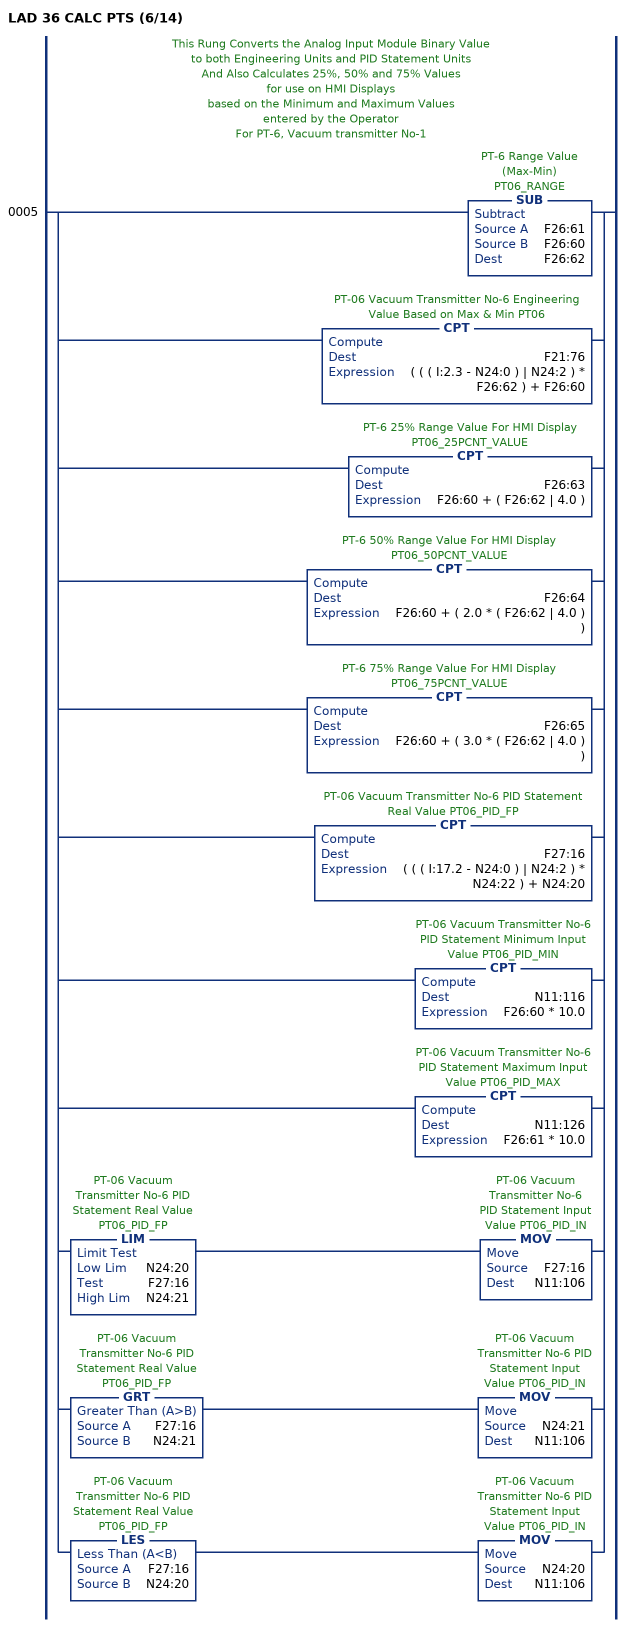
% Rung: 5 %
% This Rung Converts the Analog Input Module Binary Value
% to both Engineering Units and PID Statement Units
% And Also Calculates 25%, 50% and 75% Values
% for use on HMI Displays
% based on the Minimum and Maximum Values
% entered by the Operator
%    For PT-6, Vacuum transmitter No-1 %
SOR BST SUB F26:61 F26:60 F26:62 NXB CPT F21:76 " ( ( ( I:2.3 - N24:0 ) | N24:2 ) * F26:62 ) + F26:60 " NXB CPT F26:63 " F26:60 + ( F26:62 | 4.0 ) " NXB CPT F26:64 " F26:60 + ( 2.0 * ( F26:62 | 4.0 ) ) " NXB CPT F26:65 " F26:60 + ( 3.0 * ( F26:62 | 4.0 ) ) " NXB CPT F27:16 " ( ( ( I:17.2 - N24:0 ) | N24:2 ) * N24:22 ) + N24:20 " NXB CPT N11:116 " F26:60 * 10.0 " NXB CPT N11:126 " F26:61 * 10.0 " NXB LIM N24:20 F27:16 N24:21 MOV F27:16 N11:106 NXB GRT F27:16 N24:21 MOV N24:21 N11:106 NXB LES F27:16 N24:20 MOV N24:20 N11:106 BND EOR
%   F26:61  PT06_MAX  "PT-6 Maximum Value" %
%   F26:60  PT06_MIN  "PT-6 Minimum Value" %
%   F26:62  PT06_RANGE  "PT-6 Range Value (Max-Min)" %
%   F21:76  PT06  "PT-06 Vacuum Transmitter No-6 Engineering Value Based on Max & Min" %
%   I:2.3  PT61_BIN  "PT-6 Binary Input From Transmitter Analog Input Module" %
%   N24:0  AI_CURRENT_MIN  "Analog Input Minimum Value = 4 mA DC (From AI Module)" %
%   N24:2  AI_CURRENT_RANGE  "Analog Input Current Range Value = (AI_MAX - AI_MIN) For Use Elswhere" %
%   F26:63  PT06_25PCNT_VALUE  "PT-6 25% Range Value For HMI Display" %
%   F26:64  PT06_50PCNT_VALUE  "PT-6 50% Range Value For HMI Display" %
%   F26:65  PT06_75PCNT_VALUE  "PT-6 75% Range Value For HMI Display" %
%   F27:16  PT06_PID_FP  "PT-06 Vacuum Transmitter No-6 PID Statement Real Value" %
%   I:17.2  FT06_BIN  "FT-6 Feed Flow Binary Input From Transmitter 1 Analog Input Module" %
%   N24:22  PID_RANGE  "PID Statement Range Value = (PID_MAX - PID_MIN) For Use Elswhere" %
%   N24:20  PID_MIN  "PID Statement Minimum Value" %
%   N11:116  PT06_PID_MIN  "PT-06 Vacuum Transmitter No-6 PID Statement Minimum Input Value" %
%   N11:126  PT06_PID_MAX  "PT-06 Vacuum Transmitter No-6 PID Statement Maximum Input Value" %
%   N24:21  PID_MAX  "PID Statement Maximum Value" %
%   N11:106  PT06_PID_IN  "PT-06 Vacuum Transmitter No-6 PID Statement Input Value" %

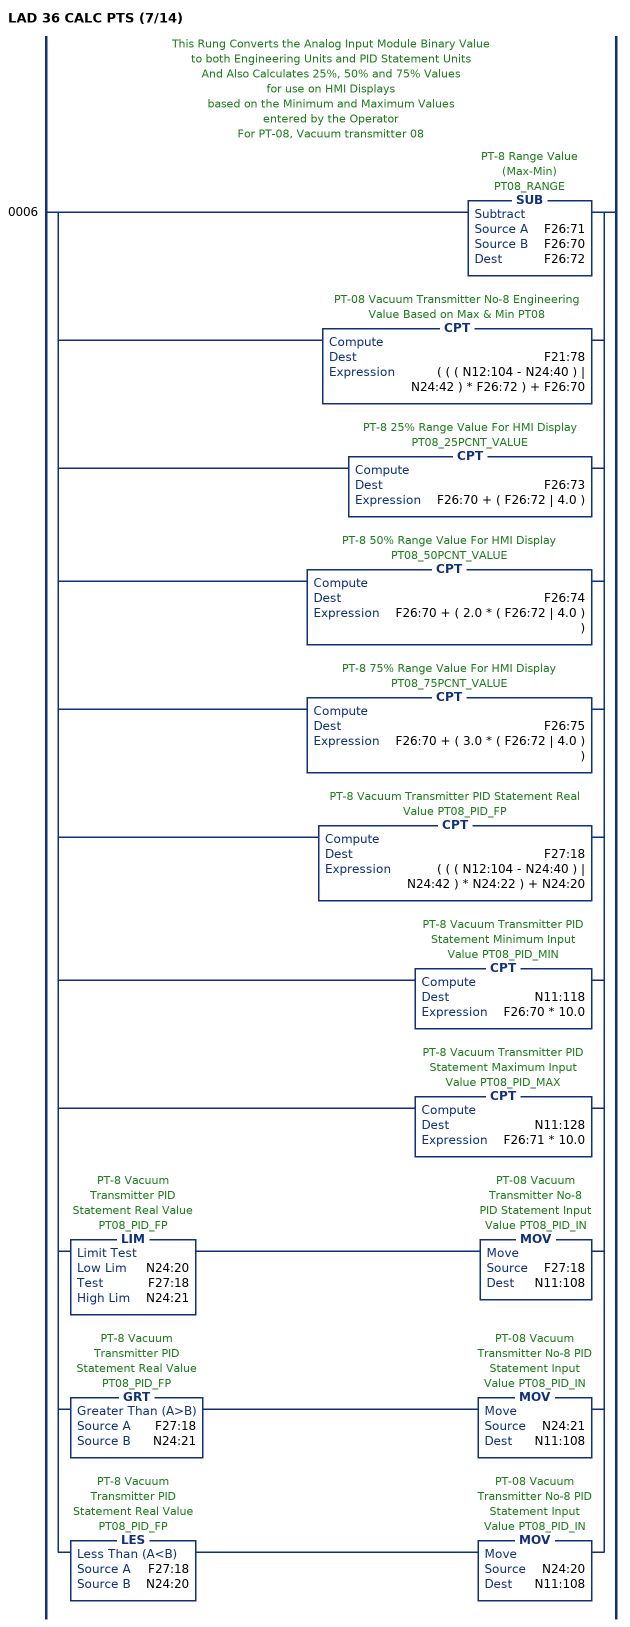
% Rung: 6 %
% This Rung Converts the Analog Input Module Binary Value
% to both Engineering Units and PID Statement Units
% And Also Calculates 25%, 50% and 75% Values
% for use on HMI Displays
% based on the Minimum and Maximum Values
% entered by the Operator
%    For PT-08, Vacuum transmitter 08 %
SOR BST SUB F26:71 F26:70 F26:72 NXB CPT F21:78 " ( ( ( N12:104 - N24:40 ) | N24:42 ) * F26:72 ) + F26:70 " NXB CPT F26:73 " F26:70 + ( F26:72 | 4.0 ) " NXB CPT F26:74 " F26:70 + ( 2.0 * ( F26:72 | 4.0 ) ) " NXB CPT F26:75 " F26:70 + ( 3.0 * ( F26:72 | 4.0 ) ) " NXB CPT F27:18 " ( ( ( N12:104 - N24:40 ) | N24:42 ) * N24:22 ) + N24:20 " NXB CPT N11:118 " F26:70 * 10.0 " NXB CPT N11:128 " F26:71 * 10.0 " NXB LIM N24:20 F27:18 N24:21 MOV F27:18 N11:108 NXB GRT F27:18 N24:21 MOV N24:21 N11:108 NXB LES F27:18 N24:20 MOV N24:20 N11:108 BND EOR
%   F26:71  PT08_MAX  "PT-8 Maximum Value" %
%   F26:70  PT08_MIN  "PT-8 Minimum Value" %
%   F26:72  PT08_RANGE  "PT-8 Range Value (Max-Min)" %
%   F21:78  PT08  "PT-08 Vacuum Transmitter No-8 Engineering Value Based on Max & Min" %
%   N12:104  AI105_BIN_DATA %
%   N24:40  AI_CURRENT_MIN_IE8  "Analog Input Minimum Value = 4 mA DC (From IE8 AI Module)" %
%   N24:42  AI_CURRENT_RANGE_IE8  "IE8 Analog Input Current Range Value = (AI_MAX - AI_MIN) For Use Elswhere" %
%   F26:73  PT08_25PCNT_VALUE  "PT-8 25% Range Value For HMI Display" %
%   F26:74  PT08_50PCNT_VALUE  "PT-8 50% Range Value For HMI Display" %
%   F26:75  PT08_75PCNT_VALUE  "PT-8 75% Range Value For HMI Display" %
%   F27:18  PT08_PID_FP  "PT-8 Vacuum Transmitter PID Statement Real Value" %
%   N24:22  PID_RANGE  "PID Statement Range Value = (PID_MAX - PID_MIN) For Use Elswhere" %
%   N24:20  PID_MIN  "PID Statement Minimum Value" %
%   N11:118  PT08_PID_MIN  "PT-8 Vacuum Transmitter PID Statement Minimum Input Value" %
%   N11:128  PT08_PID_MAX  "PT-8 Vacuum Transmitter PID Statement Maximum Input Value" %
%   N24:21  PID_MAX  "PID Statement Maximum Value" %
%   N11:108  PT08_PID_IN  "PT-08 Vacuum Transmitter No-8 PID Statement Input Value" %

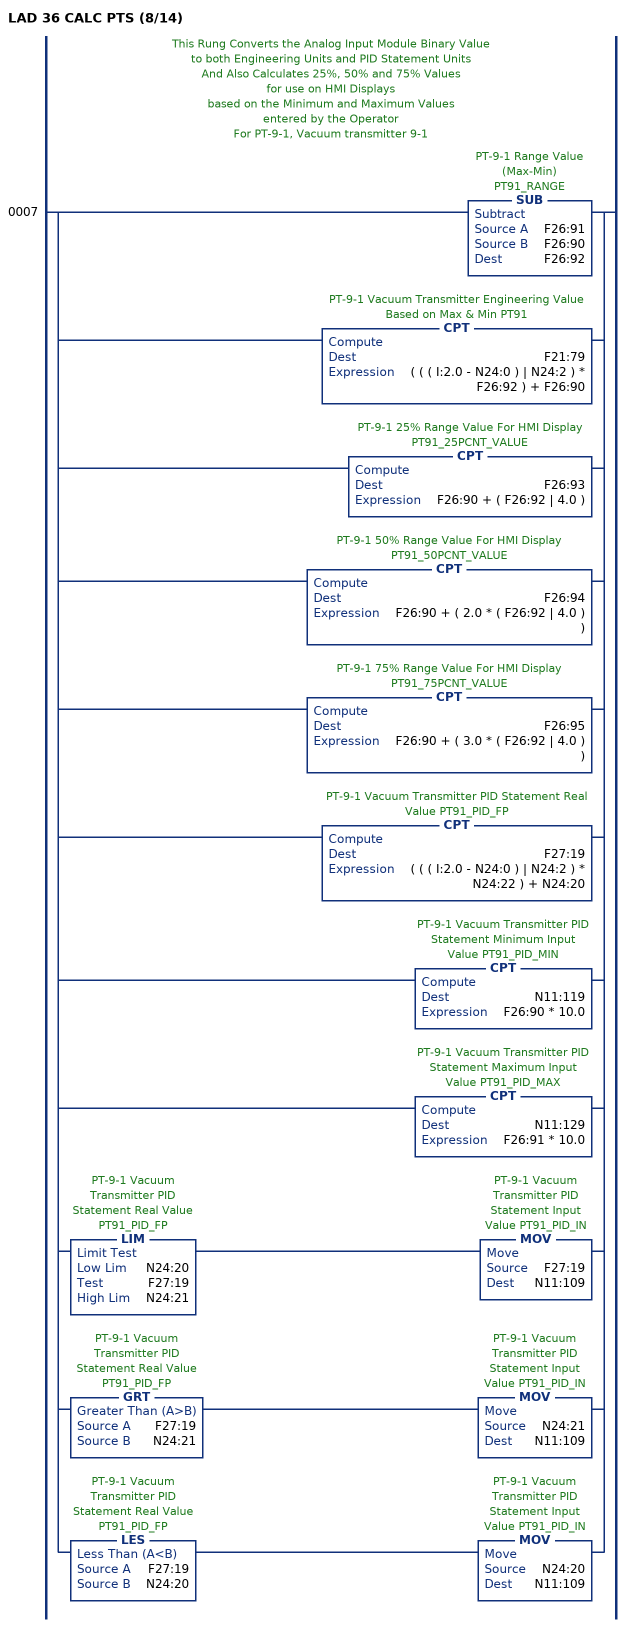
% Rung: 7 %
% This Rung Converts the Analog Input Module Binary Value
% to both Engineering Units and PID Statement Units
% And Also Calculates 25%, 50% and 75% Values
% for use on HMI Displays
% based on the Minimum and Maximum Values
% entered by the Operator
%    For PT-9-1, Vacuum transmitter 9-1 %
SOR BST SUB F26:91 F26:90 F26:92 NXB CPT F21:79 " ( ( ( I:2.0 - N24:0 ) | N24:2 ) * F26:92 ) + F26:90 " NXB CPT F26:93 " F26:90 + ( F26:92 | 4.0 ) " NXB CPT F26:94 " F26:90 + ( 2.0 * ( F26:92 | 4.0 ) ) " NXB CPT F26:95 " F26:90 + ( 3.0 * ( F26:92 | 4.0 ) ) " NXB CPT F27:19 " ( ( ( I:2.0 - N24:0 ) | N24:2 ) * N24:22 ) + N24:20 " NXB CPT N11:119 " F26:90 * 10.0 " NXB CPT N11:129 " F26:91 * 10.0 " NXB LIM N24:20 F27:19 N24:21 MOV F27:19 N11:109 NXB GRT F27:19 N24:21 MOV N24:21 N11:109 NXB LES F27:19 N24:20 MOV N24:20 N11:109 BND EOR
%   F26:91  PT91_MAX  "PT-9-1 Maximum Value" %
%   F26:90  PT91_MIN  "PT-9-1 Minimum Value" %
%   F26:92  PT91_RANGE  "PT-9-1 Range Value (Max-Min)" %
%   F21:79  PT91  "PT-9-1 Vacuum Transmitter Engineering Value Based on Max & Min" %
%   I:2.0  PT91_BIN  "PT-9-1 Binary Input From Transmitter Analog Input Module" %
%   N24:0  AI_CURRENT_MIN  "Analog Input Minimum Value = 4 mA DC (From AI Module)" %
%   N24:2  AI_CURRENT_RANGE  "Analog Input Current Range Value = (AI_MAX - AI_MIN) For Use Elswhere" %
%   F26:93  PT91_25PCNT_VALUE  "PT-9-1 25% Range Value For HMI Display" %
%   F26:94  PT91_50PCNT_VALUE  "PT-9-1 50% Range Value For HMI Display" %
%   F26:95  PT91_75PCNT_VALUE  "PT-9-1 75% Range Value For HMI Display" %
%   F27:19  PT91_PID_FP  "PT-9-1 Vacuum Transmitter PID Statement Real Value" %
%   N24:22  PID_RANGE  "PID Statement Range Value = (PID_MAX - PID_MIN) For Use Elswhere" %
%   N24:20  PID_MIN  "PID Statement Minimum Value" %
%   N11:119  PT91_PID_MIN  "PT-9-1 Vacuum Transmitter PID Statement Minimum Input Value" %
%   N11:129  PT91_PID_MAX  "PT-9-1 Vacuum Transmitter PID Statement Maximum Input Value" %
%   N24:21  PID_MAX  "PID Statement Maximum Value" %
%   N11:109  PT91_PID_IN  "PT-9-1 Vacuum Transmitter PID Statement Input Value" %

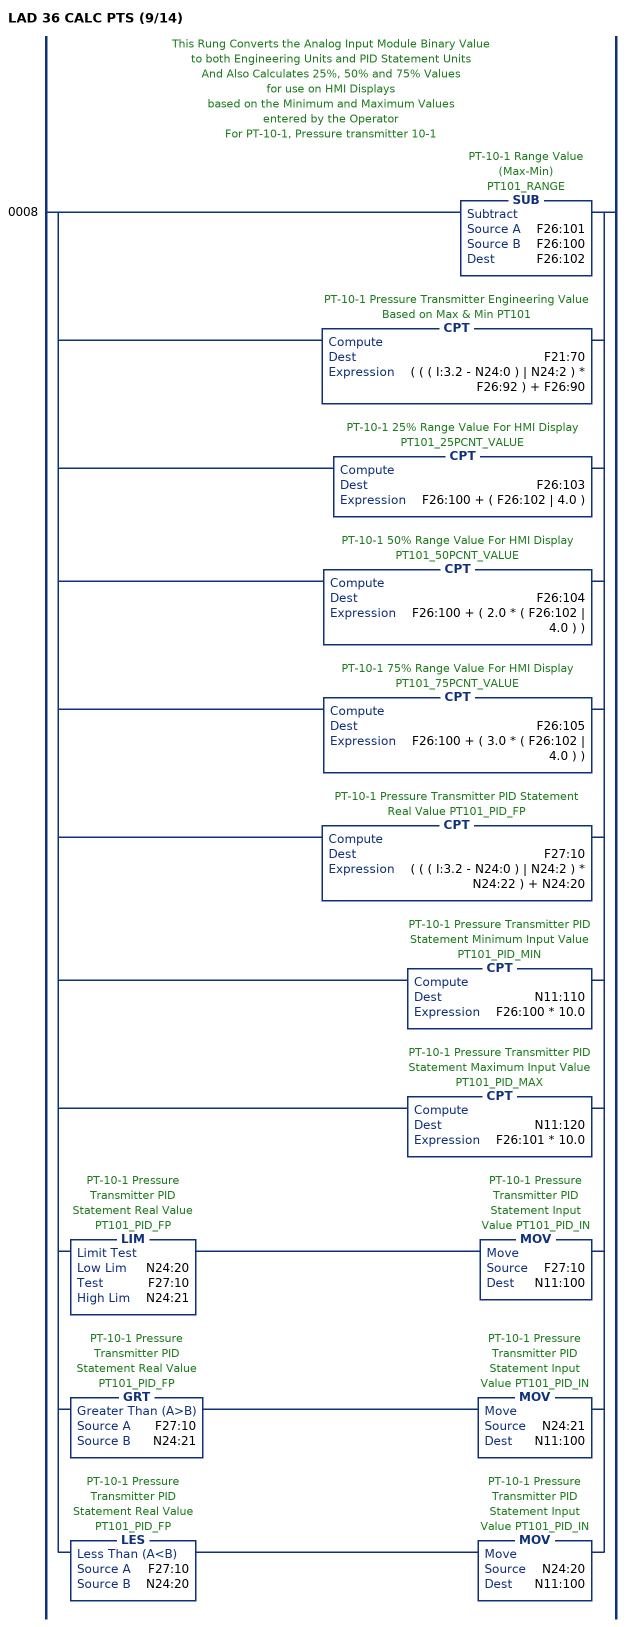
% Rung: 8 %
% This Rung Converts the Analog Input Module Binary Value
% to both Engineering Units and PID Statement Units
% And Also Calculates 25%, 50% and 75% Values
% for use on HMI Displays
% based on the Minimum and Maximum Values
% entered by the Operator
%    For PT-10-1, Pressure transmitter 10-1 %
SOR BST SUB F26:101 F26:100 F26:102 NXB CPT F21:70 " ( ( ( I:3.2 - N24:0 ) | N24:2 ) * F26:92 ) + F26:90 " NXB CPT F26:103 " F26:100 + ( F26:102 | 4.0 ) " NXB CPT F26:104 " F26:100 + ( 2.0 * ( F26:102 | 4.0 ) ) " NXB CPT F26:105 " F26:100 + ( 3.0 * ( F26:102 | 4.0 ) ) " NXB CPT F27:10 " ( ( ( I:3.2 - N24:0 ) | N24:2 ) * N24:22 ) + N24:20 " NXB CPT N11:110 " F26:100 * 10.0 " NXB CPT N11:120 " F26:101 * 10.0 " NXB LIM N24:20 F27:10 N24:21 MOV F27:10 N11:100 NXB GRT F27:10 N24:21 MOV N24:21 N11:100 NXB LES F27:10 N24:20 MOV N24:20 N11:100 BND EOR
%   F26:101  PT101_MAX  "PT-10-1 Maximum Value" %
%   F26:100  PT101_MIN  "PT-10-1 Minimum Value" %
%   F26:102  PT101_RANGE  "PT-10-1 Range Value (Max-Min)" %
%   F21:70  PT101  "PT-10-1 Pressure Transmitter Engineering Value Based on Max & Min" %
%   I:3.2  PT101_BIN  "PT-10-1 Press Binary Input From Transmitter Analog Input Module" %
%   N24:0  AI_CURRENT_MIN  "Analog Input Minimum Value = 4 mA DC (From AI Module)" %
%   N24:2  AI_CURRENT_RANGE  "Analog Input Current Range Value = (AI_MAX - AI_MIN) For Use Elswhere" %
%   F26:92  PT91_RANGE  "PT-9-1 Range Value (Max-Min)" %
%   F26:90  PT91_MIN  "PT-9-1 Minimum Value" %
%   F26:103  PT101_25PCNT_VALUE  "PT-10-1 25% Range Value For HMI Display" %
%   F26:104  PT101_50PCNT_VALUE  "PT-10-1 50% Range Value For HMI Display" %
%   F26:105  PT101_75PCNT_VALUE  "PT-10-1 75% Range Value For HMI Display" %
%   F27:10  PT101_PID_FP  "PT-10-1 Pressure Transmitter PID Statement Real Value" %
%   N24:22  PID_RANGE  "PID Statement Range Value = (PID_MAX - PID_MIN) For Use Elswhere" %
%   N24:20  PID_MIN  "PID Statement Minimum Value" %
%   N11:110  PT101_PID_MIN  "PT-10-1 Pressure Transmitter PID Statement Minimum Input Value" %
%   N11:120  PT101_PID_MAX  "PT-10-1 Pressure Transmitter PID Statement Maximum Input Value" %
%   N24:21  PID_MAX  "PID Statement Maximum Value" %
%   N11:100  PT101_PID_IN  "PT-10-1 Pressure Transmitter PID Statement Input Value" %

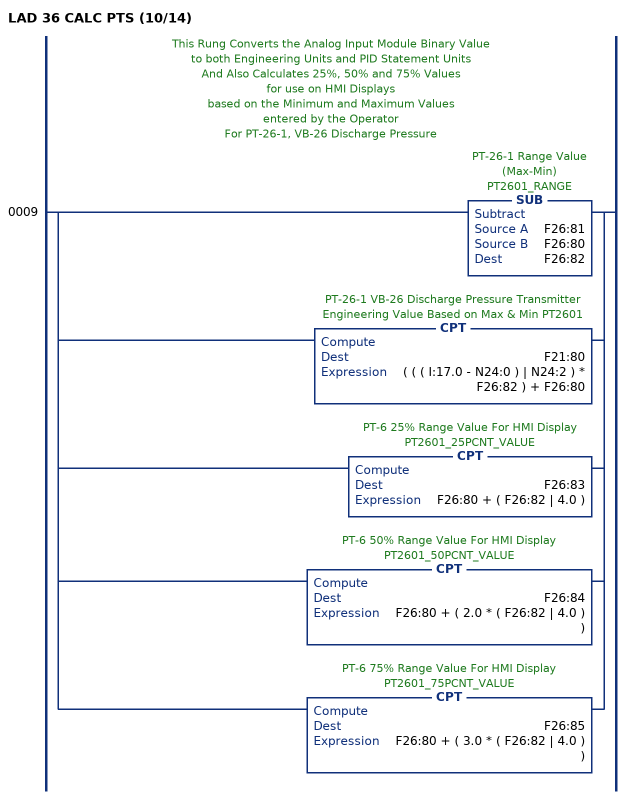
% Rung: 9 %
% This Rung Converts the Analog Input Module Binary Value
% to both Engineering Units and PID Statement Units
% And Also Calculates 25%, 50% and 75% Values
% for use on HMI Displays
% based on the Minimum and Maximum Values
% entered by the Operator
%    For PT-26-1, VB-26 Discharge Pressure %
SOR BST SUB F26:81 F26:80 F26:82 NXB CPT F21:80 " ( ( ( I:17.0 - N24:0 ) | N24:2 ) * F26:82 ) + F26:80 " NXB CPT F26:83 " F26:80 + ( F26:82 | 4.0 ) " NXB CPT F26:84 " F26:80 + ( 2.0 * ( F26:82 | 4.0 ) ) " NXB CPT F26:85 " F26:80 + ( 3.0 * ( F26:82 | 4.0 ) ) " BND EOR
%   F26:81  PT2601_MAX  "PT-6 Maximum Value" %
%   F26:80  PT2601_MIN  "PT-6 Minimum Value" %
%   F26:82  PT2601_RANGE  "PT-26-1 Range Value (Max-Min)" %
%   F21:80  PT2601  "PT-26-1 VB-26 Discharge Pressure Transmitter Engineering Value Based on Max & Min" %
%   I:17.0  LIT01_BIN  "LIT-1 Binary Input From Transmitter Analog Input Module" %
%   N24:0  AI_CURRENT_MIN  "Analog Input Minimum Value = 4 mA DC (From AI Module)" %
%   N24:2  AI_CURRENT_RANGE  "Analog Input Current Range Value = (AI_MAX - AI_MIN) For Use Elswhere" %
%   F26:83  PT2601_25PCNT_VALUE  "PT-6 25% Range Value For HMI Display" %
%   F26:84  PT2601_50PCNT_VALUE  "PT-6 50% Range Value For HMI Display" %
%   F26:85  PT2601_75PCNT_VALUE  "PT-6 75% Range Value For HMI Display" %

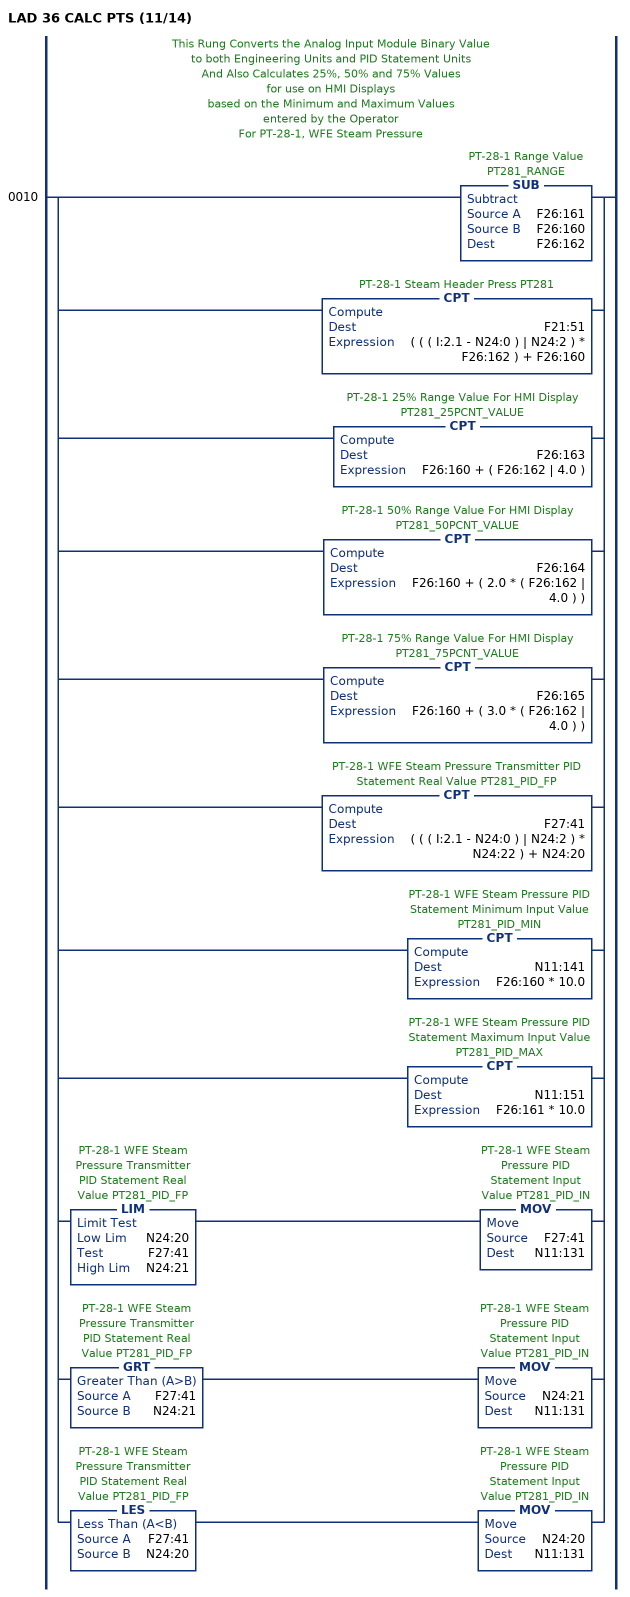
% Rung: 10 %
% This Rung Converts the Analog Input Module Binary Value
% to both Engineering Units and PID Statement Units
% And Also Calculates 25%, 50% and 75% Values
% for use on HMI Displays
% based on the Minimum and Maximum Values
% entered by the Operator
%    For PT-28-1, WFE Steam Pressure %
SOR BST SUB F26:161 F26:160 F26:162 NXB CPT F21:51 " ( ( ( I:2.1 - N24:0 ) | N24:2 ) * F26:162 ) + F26:160 " NXB CPT F26:163 " F26:160 + ( F26:162 | 4.0 ) " NXB CPT F26:164 " F26:160 + ( 2.0 * ( F26:162 | 4.0 ) ) " NXB CPT F26:165 " F26:160 + ( 3.0 * ( F26:162 | 4.0 ) ) " NXB CPT F27:41 " ( ( ( I:2.1 - N24:0 ) | N24:2 ) * N24:22 ) + N24:20 " NXB CPT N11:141 " F26:160 * 10.0 " NXB CPT N11:151 " F26:161 * 10.0 " NXB LIM N24:20 F27:41 N24:21 MOV F27:41 N11:131 NXB GRT F27:41 N24:21 MOV N24:21 N11:131 NXB LES F27:41 N24:20 MOV N24:20 N11:131 BND EOR
%   F26:161  PT281_MAX  "PT-28-1 Maximum Value" %
%   F26:160  PT281_MIN  "PT-28-1 Minimum Value" %
%   F26:162  PT281_RANGE  "PT-28-1 Range Value" %
%   F21:51  PT281  "PT-28-1 Steam Header Press" %
%   I:2.1  PT281_BIN  "PT-28-1 Steam Header Press Binary Input From Transmitter Analog Input Module" %
%   N24:0  AI_CURRENT_MIN  "Analog Input Minimum Value = 4 mA DC (From AI Module)" %
%   N24:2  AI_CURRENT_RANGE  "Analog Input Current Range Value = (AI_MAX - AI_MIN) For Use Elswhere" %
%   F26:163  PT281_25PCNT_VALUE  "PT-28-1 25% Range Value For HMI Display" %
%   F26:164  PT281_50PCNT_VALUE  "PT-28-1 50% Range Value For HMI Display" %
%   F26:165  PT281_75PCNT_VALUE  "PT-28-1 75% Range Value For HMI Display" %
%   F27:41  PT281_PID_FP  "PT-28-1 WFE Steam Pressure Transmitter PID Statement Real Value" %
%   N24:22  PID_RANGE  "PID Statement Range Value = (PID_MAX - PID_MIN) For Use Elswhere" %
%   N24:20  PID_MIN  "PID Statement Minimum Value" %
%   N11:141  PT281_PID_MIN  "PT-28-1 WFE Steam Pressure PID Statement Minimum Input Value" %
%   N11:151  PT281_PID_MAX  "PT-28-1 WFE Steam Pressure PID Statement Maximum Input Value" %
%   N24:21  PID_MAX  "PID Statement Maximum Value" %
%   N11:131  PT281_PID_IN  "PT-28-1 WFE Steam Pressure PID Statement Input Value" %

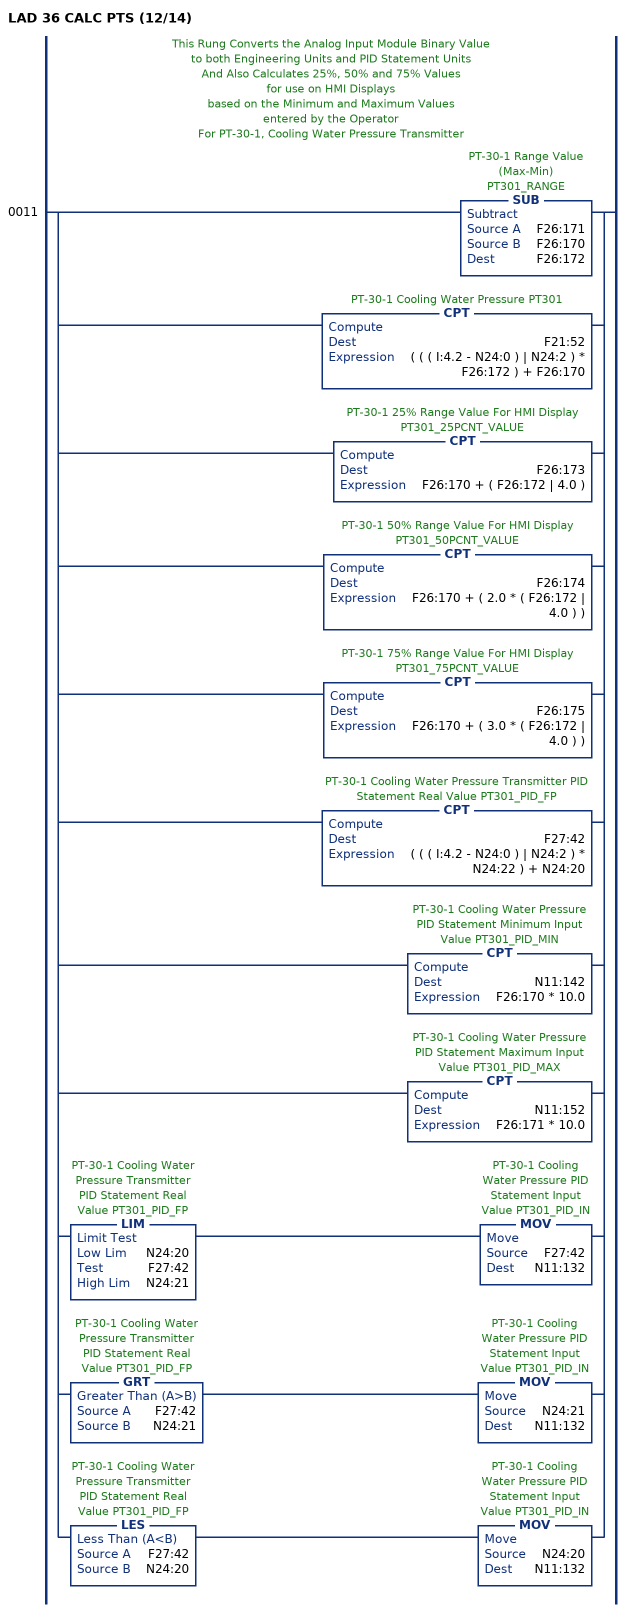
% Rung: 11 %
% This Rung Converts the Analog Input Module Binary Value
% to both Engineering Units and PID Statement Units
% And Also Calculates 25%, 50% and 75% Values
% for use on HMI Displays
% based on the Minimum and Maximum Values
% entered by the Operator
%    For PT-30-1, Cooling Water Pressure Transmitter %
SOR BST SUB F26:171 F26:170 F26:172 NXB CPT F21:52 " ( ( ( I:4.2 - N24:0 ) | N24:2 ) * F26:172 ) + F26:170 " NXB CPT F26:173 " F26:170 + ( F26:172 | 4.0 ) " NXB CPT F26:174 " F26:170 + ( 2.0 * ( F26:172 | 4.0 ) ) " NXB CPT F26:175 " F26:170 + ( 3.0 * ( F26:172 | 4.0 ) ) " NXB CPT F27:42 " ( ( ( I:4.2 - N24:0 ) | N24:2 ) * N24:22 ) + N24:20 " NXB CPT N11:142 " F26:170 * 10.0 " NXB CPT N11:152 " F26:171 * 10.0 " NXB LIM N24:20 F27:42 N24:21 MOV F27:42 N11:132 NXB GRT F27:42 N24:21 MOV N24:21 N11:132 NXB LES F27:42 N24:20 MOV N24:20 N11:132 BND EOR
%   F26:171  PT301_MAX  "PT-30-1 Maximum Value" %
%   F26:170  PT301_MIN  "PT-30-1 Minimum Value" %
%   F26:172  PT301_RANGE  "PT-30-1 Range Value (Max-Min)" %
%   F21:52  PT301  "PT-30-1 Cooling Water Pressure" %
%   I:4.2  PT301_BIN  "PT-30-1 City Water Supply Header Pressure" %
%   N24:0  AI_CURRENT_MIN  "Analog Input Minimum Value = 4 mA DC (From AI Module)" %
%   N24:2  AI_CURRENT_RANGE  "Analog Input Current Range Value = (AI_MAX - AI_MIN) For Use Elswhere" %
%   F26:173  PT301_25PCNT_VALUE  "PT-30-1 25% Range Value For HMI Display" %
%   F26:174  PT301_50PCNT_VALUE  "PT-30-1 50% Range Value For HMI Display" %
%   F26:175  PT301_75PCNT_VALUE  "PT-30-1 75% Range Value For HMI Display" %
%   F27:42  PT301_PID_FP  "PT-30-1 Cooling Water Pressure Transmitter PID Statement Real Value" %
%   N24:22  PID_RANGE  "PID Statement Range Value = (PID_MAX - PID_MIN) For Use Elswhere" %
%   N24:20  PID_MIN  "PID Statement Minimum Value" %
%   N11:142  PT301_PID_MIN  "PT-30-1 Cooling Water Pressure PID Statement Minimum Input Value" %
%   N11:152  PT301_PID_MAX  "PT-30-1 Cooling Water Pressure PID Statement Maximum Input Value" %
%   N24:21  PID_MAX  "PID Statement Maximum Value" %
%   N11:132  PT301_PID_IN  "PT-30-1 Cooling Water Pressure PID Statement Input Value" %

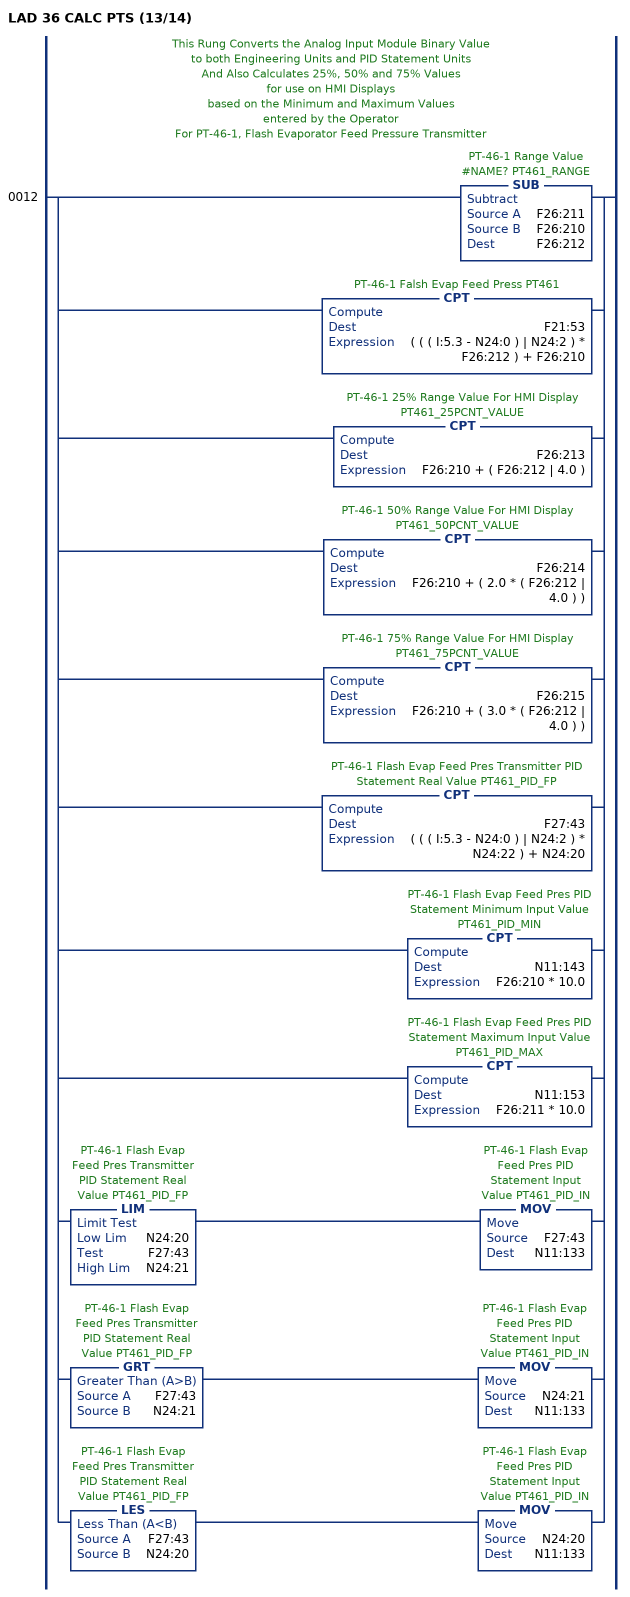
% Rung: 12 %
% This Rung Converts the Analog Input Module Binary Value
% to both Engineering Units and PID Statement Units
% And Also Calculates 25%, 50% and 75% Values
% for use on HMI Displays
% based on the Minimum and Maximum Values
% entered by the Operator
%    For PT-46-1, Flash Evaporator Feed Pressure Transmitter %
SOR BST SUB F26:211 F26:210 F26:212 NXB CPT F21:53 " ( ( ( I:5.3 - N24:0 ) | N24:2 ) * F26:212 ) + F26:210 " NXB CPT F26:213 " F26:210 + ( F26:212 | 4.0 ) " NXB CPT F26:214 " F26:210 + ( 2.0 * ( F26:212 | 4.0 ) ) " NXB CPT F26:215 " F26:210 + ( 3.0 * ( F26:212 | 4.0 ) ) " NXB CPT F27:43 " ( ( ( I:5.3 - N24:0 ) | N24:2 ) * N24:22 ) + N24:20 " NXB CPT N11:143 " F26:210 * 10.0 " NXB CPT N11:153 " F26:211 * 10.0 " NXB LIM N24:20 F27:43 N24:21 MOV F27:43 N11:133 NXB GRT F27:43 N24:21 MOV N24:21 N11:133 NXB LES F27:43 N24:20 MOV N24:20 N11:133 BND EOR
%   F26:211  PT461_MAX  "PT-46-1 Maximum Value" %
%   F26:210  PT461_MIN  "PT-46-1 Minimum Value" %
%   F26:212  PT461_RANGE  "PT-46-1 Range Value #NAME?" %
%   F21:53  PT461  "PT-46-1 Falsh Evap Feed Press" %
%   I:5.3  PT461_BIN  "PT-46-1 Flash Evap Feed Pres Binary Input From Transmitter Analog Input Module" %
%   N24:0  AI_CURRENT_MIN  "Analog Input Minimum Value = 4 mA DC (From AI Module)" %
%   N24:2  AI_CURRENT_RANGE  "Analog Input Current Range Value = (AI_MAX - AI_MIN) For Use Elswhere" %
%   F26:213  PT461_25PCNT_VALUE  "PT-46-1 25% Range Value For HMI Display" %
%   F26:214  PT461_50PCNT_VALUE  "PT-46-1 50% Range Value For HMI Display" %
%   F26:215  PT461_75PCNT_VALUE  "PT-46-1 75% Range Value For HMI Display" %
%   F27:43  PT461_PID_FP  "PT-46-1 Flash Evap Feed Pres Transmitter PID Statement Real Value" %
%   N24:22  PID_RANGE  "PID Statement Range Value = (PID_MAX - PID_MIN) For Use Elswhere" %
%   N24:20  PID_MIN  "PID Statement Minimum Value" %
%   N11:143  PT461_PID_MIN  "PT-46-1 Flash Evap Feed Pres PID Statement Minimum Input Value" %
%   N11:153  PT461_PID_MAX  "PT-46-1 Flash Evap Feed Pres PID Statement Maximum Input Value" %
%   N24:21  PID_MAX  "PID Statement Maximum Value" %
%   N11:133  PT461_PID_IN  "PT-46-1 Flash Evap Feed Pres PID Statement Input Value" %

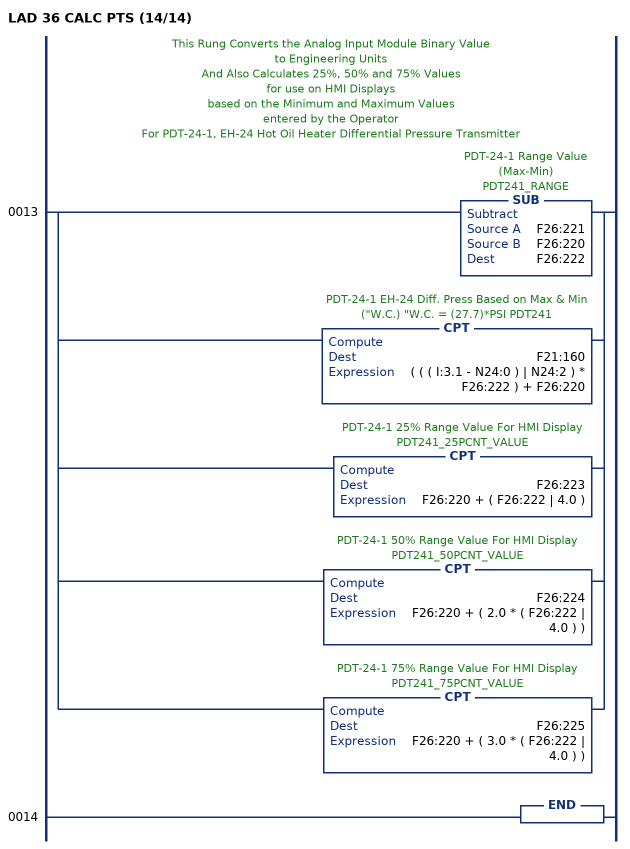
% Rung: 13 %
% This Rung Converts the Analog Input Module Binary Value
% to Engineering Units
% And Also Calculates 25%, 50% and 75% Values
% for use on HMI Displays
% based on the Minimum and Maximum Values
% entered by the Operator
%    For PDT-24-1, EH-24 Hot Oil Heater Differential Pressure Transmitter %
SOR BST SUB F26:221 F26:220 F26:222 NXB CPT F21:160 " ( ( ( I:3.1 - N24:0 ) | N24:2 ) * F26:222 ) + F26:220 " NXB CPT F26:223 " F26:220 + ( F26:222 | 4.0 ) " NXB CPT F26:224 " F26:220 + ( 2.0 * ( F26:222 | 4.0 ) ) " NXB CPT F26:225 " F26:220 + ( 3.0 * ( F26:222 | 4.0 ) ) " BND EOR
%   F26:221  PDT241_MAX  "PDT-24-1 Maximum Value" %
%   F26:220  PDT241_MIN  "PDT-24-1 Minimum Value" %
%   F26:222  PDT241_RANGE  "PDT-24-1 Range Value (Max-Min)" %
%   F21:160  PDT241  "PDT-24-1 EH-24 Diff. Press Based on Max & Min ("W.C.) "W.C. = (27.7)*PSI" %
%   I:3.1  PDT241_BIN  "PDT-24-1 EH-24 Diff Press Input (BIN)" %
%   N24:0  AI_CURRENT_MIN  "Analog Input Minimum Value = 4 mA DC (From AI Module)" %
%   N24:2  AI_CURRENT_RANGE  "Analog Input Current Range Value = (AI_MAX - AI_MIN) For Use Elswhere" %
%   F26:223  PDT241_25PCNT_VALUE  "PDT-24-1 25% Range Value For HMI Display" %
%   F26:224  PDT241_50PCNT_VALUE  "PDT-24-1 50% Range Value For HMI Display" %
%   F26:225  PDT241_75PCNT_VALUE  "PDT-24-1 75% Range Value For HMI Display" %
% Rung: 14 %
SOR END EOR

LADDER 37 "CALC FTS"    % Calculate FT's Based on Max & Min Ranges %
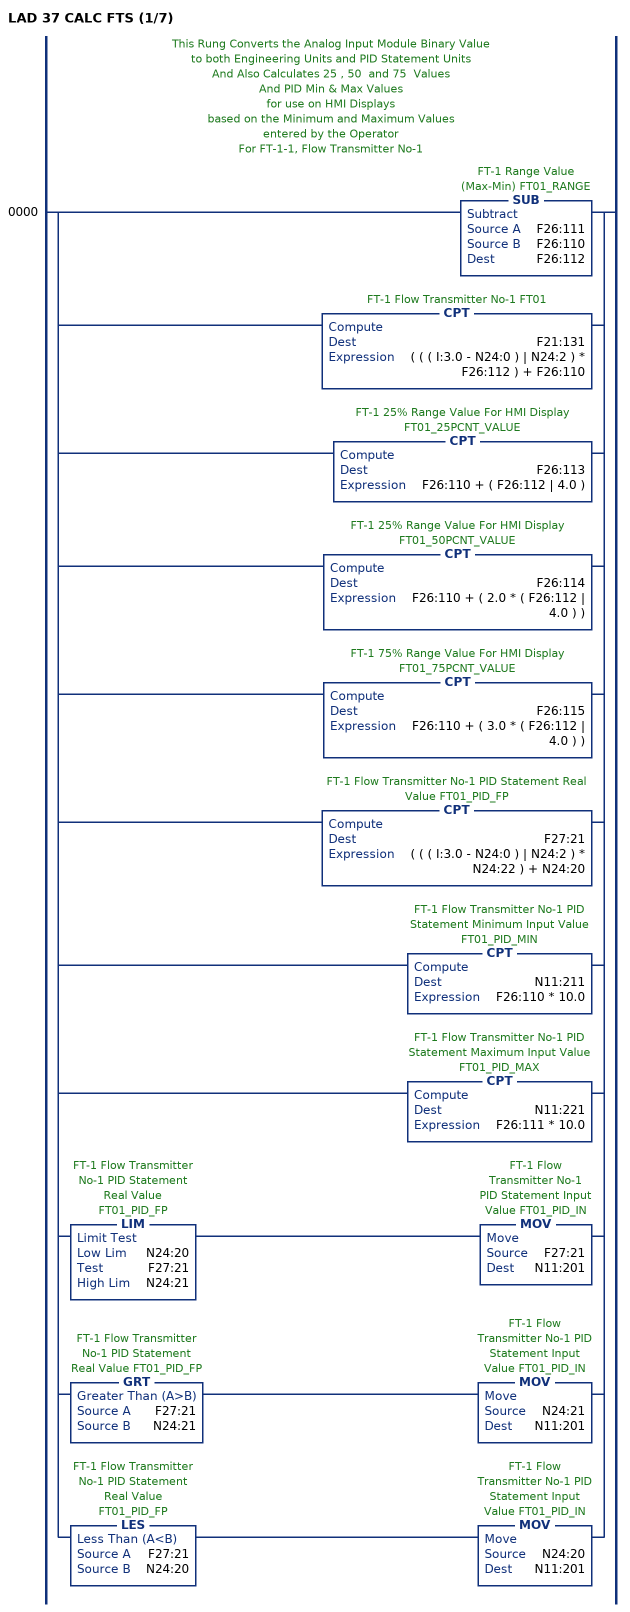
% Rung: 0 %
% This Rung Converts the Analog Input Module Binary Value
% to both Engineering Units and PID Statement Units
% And Also Calculates 25 , 50  and 75  Values
% And PID Min & Max Values
% for use on HMI Displays
% based on the Minimum and Maximum Values
% entered by the Operator
%    For FT-1-1, Flow Transmitter No-1 %
SOR BST SUB F26:111 F26:110 F26:112 NXB CPT F21:131 " ( ( ( I:3.0 - N24:0 ) | N24:2 ) * F26:112 ) + F26:110 " NXB CPT F26:113 " F26:110 + ( F26:112 | 4.0 ) " NXB CPT F26:114 " F26:110 + ( 2.0 * ( F26:112 | 4.0 ) ) " NXB CPT F26:115 " F26:110 + ( 3.0 * ( F26:112 | 4.0 ) ) " NXB CPT F27:21 " ( ( ( I:3.0 - N24:0 ) | N24:2 ) * N24:22 ) + N24:20 " NXB CPT N11:211 " F26:110 * 10.0 " NXB CPT N11:221 " F26:111 * 10.0 " NXB LIM N24:20 F27:21 N24:21 MOV F27:21 N11:201 NXB GRT F27:21 N24:21 MOV N24:21 N11:201 NXB LES F27:21 N24:20 MOV N24:20 N11:201 BND EOR
%   F26:111  FT01_MAX  "FT-1 Maximum Value" %
%   F26:110  FT01_MIN  "FT-1 Minimum Value" %
%   F26:112  FT01_RANGE  "FT-1 Range Value (Max-Min)" %
%   F21:131  FT01  "FT-1 Flow Transmitter No-1" %
%   I:3.0  FT01_BIN  "FT-1 Feed Flow Binary Input From Transmitter 1 Analog Input Module" %
%   N24:0  AI_CURRENT_MIN  "Analog Input Minimum Value = 4 mA DC (From AI Module)" %
%   N24:2  AI_CURRENT_RANGE  "Analog Input Current Range Value = (AI_MAX - AI_MIN) For Use Elswhere" %
%   F26:113  FT01_25PCNT_VALUE  "FT-1 25% Range Value For HMI Display" %
%   F26:114  FT01_50PCNT_VALUE  "FT-1 25% Range Value For HMI Display" %
%   F26:115  FT01_75PCNT_VALUE  "FT-1 75% Range Value For HMI Display" %
%   F27:21  FT01_PID_FP  "FT-1 Flow Transmitter No-1 PID Statement Real Value" %
%   N24:22  PID_RANGE  "PID Statement Range Value = (PID_MAX - PID_MIN) For Use Elswhere" %
%   N24:20  PID_MIN  "PID Statement Minimum Value" %
%   N11:211  FT01_PID_MIN  "FT-1 Flow Transmitter No-1 PID Statement Minimum Input Value" %
%   N11:221  FT01_PID_MAX  "FT-1 Flow Transmitter No-1 PID Statement Maximum Input Value" %
%   N24:21  PID_MAX  "PID Statement Maximum Value" %
%   N11:201  FT01_PID_IN  "FT-1 Flow Transmitter No-1 PID Statement Input Value" %

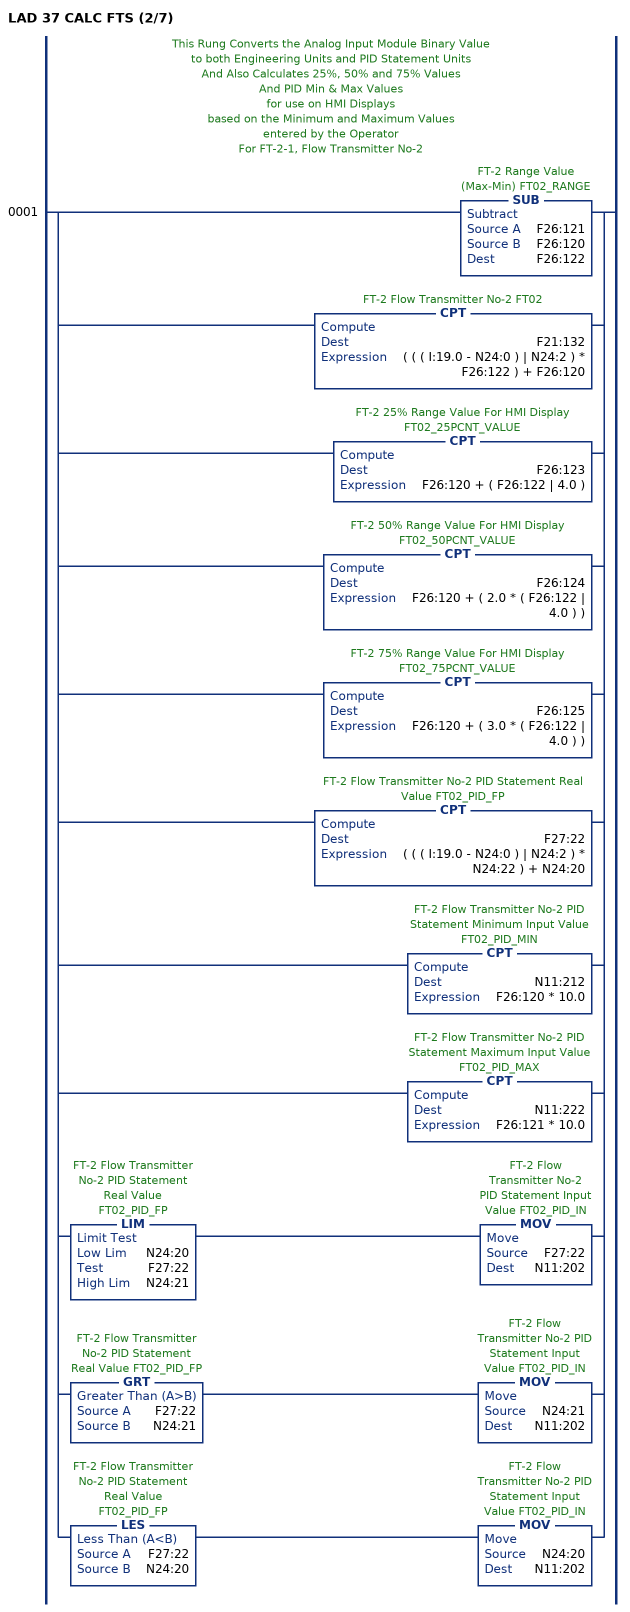
% Rung: 1 %
% This Rung Converts the Analog Input Module Binary Value
% to both Engineering Units and PID Statement Units
% And Also Calculates 25%, 50% and 75% Values
% And PID Min & Max Values
% for use on HMI Displays
% based on the Minimum and Maximum Values
% entered by the Operator
%    For FT-2-1, Flow Transmitter No-2 %
SOR BST SUB F26:121 F26:120 F26:122 NXB CPT F21:132 " ( ( ( I:19.0 - N24:0 ) | N24:2 ) * F26:122 ) + F26:120 " NXB CPT F26:123 " F26:120 + ( F26:122 | 4.0 ) " NXB CPT F26:124 " F26:120 + ( 2.0 * ( F26:122 | 4.0 ) ) " NXB CPT F26:125 " F26:120 + ( 3.0 * ( F26:122 | 4.0 ) ) " NXB CPT F27:22 " ( ( ( I:19.0 - N24:0 ) | N24:2 ) * N24:22 ) + N24:20 " NXB CPT N11:212 " F26:120 * 10.0 " NXB CPT N11:222 " F26:121 * 10.0 " NXB LIM N24:20 F27:22 N24:21 MOV F27:22 N11:202 NXB GRT F27:22 N24:21 MOV N24:21 N11:202 NXB LES F27:22 N24:20 MOV N24:20 N11:202 BND EOR
%   F26:121  FT02_MAX  "FT-2 Maximum Value" %
%   F26:120  FT02_MIN  "FT-2 Minimum Value" %
%   F26:122  FT02_RANGE  "FT-2 Range Value (Max-Min)" %
%   F21:132  FT02  "FT-2 Flow Transmitter No-2" %
%   I:19.0  FT02_BIN  "FT-2 Portable Mass Flowmeter No-2" %
%   N24:0  AI_CURRENT_MIN  "Analog Input Minimum Value = 4 mA DC (From AI Module)" %
%   N24:2  AI_CURRENT_RANGE  "Analog Input Current Range Value = (AI_MAX - AI_MIN) For Use Elswhere" %
%   F26:123  FT02_25PCNT_VALUE  "FT-2 25% Range Value For HMI Display" %
%   F26:124  FT02_50PCNT_VALUE  "FT-2 50% Range Value For HMI Display" %
%   F26:125  FT02_75PCNT_VALUE  "FT-2 75% Range Value For HMI Display" %
%   F27:22  FT02_PID_FP  "FT-2 Flow Transmitter No-2 PID Statement Real Value" %
%   N24:22  PID_RANGE  "PID Statement Range Value = (PID_MAX - PID_MIN) For Use Elswhere" %
%   N24:20  PID_MIN  "PID Statement Minimum Value" %
%   N11:212  FT02_PID_MIN  "FT-2 Flow Transmitter No-2 PID Statement Minimum Input Value" %
%   N11:222  FT02_PID_MAX  "FT-2 Flow Transmitter No-2 PID Statement Maximum Input Value" %
%   N24:21  PID_MAX  "PID Statement Maximum Value" %
%   N11:202  FT02_PID_IN  "FT-2 Flow Transmitter No-2 PID Statement Input Value" %

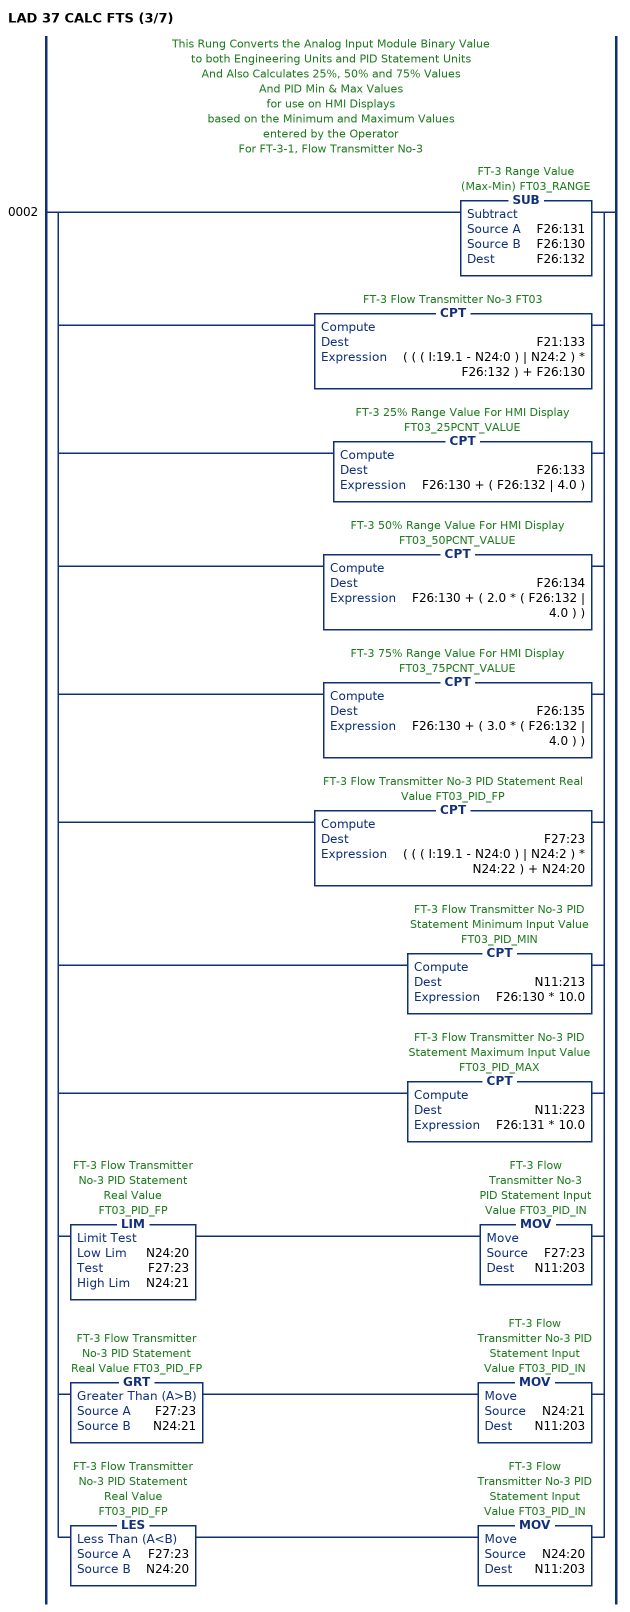
% Rung: 2 %
% This Rung Converts the Analog Input Module Binary Value
% to both Engineering Units and PID Statement Units
% And Also Calculates 25%, 50% and 75% Values
% And PID Min & Max Values
% for use on HMI Displays
% based on the Minimum and Maximum Values
% entered by the Operator
%    For FT-3-1, Flow Transmitter No-3 %
SOR BST SUB F26:131 F26:130 F26:132 NXB CPT F21:133 " ( ( ( I:19.1 - N24:0 ) | N24:2 ) * F26:132 ) + F26:130 " NXB CPT F26:133 " F26:130 + ( F26:132 | 4.0 ) " NXB CPT F26:134 " F26:130 + ( 2.0 * ( F26:132 | 4.0 ) ) " NXB CPT F26:135 " F26:130 + ( 3.0 * ( F26:132 | 4.0 ) ) " NXB CPT F27:23 " ( ( ( I:19.1 - N24:0 ) | N24:2 ) * N24:22 ) + N24:20 " NXB CPT N11:213 " F26:130 * 10.0 " NXB CPT N11:223 " F26:131 * 10.0 " NXB LIM N24:20 F27:23 N24:21 MOV F27:23 N11:203 NXB GRT F27:23 N24:21 MOV N24:21 N11:203 NXB LES F27:23 N24:20 MOV N24:20 N11:203 BND EOR
%   F26:131  FT03_MAX  "FT-3 Maximum Value" %
%   F26:130  FT03_MIN  "FT-3 Minimum Value" %
%   F26:132  FT03_RANGE  "FT-3 Range Value (Max-Min)" %
%   F21:133  FT03  "FT-3 Flow Transmitter No-3" %
%   I:19.1  FT03_BIN  "FT-3 Portable Mass Flowmeter No-3" %
%   N24:0  AI_CURRENT_MIN  "Analog Input Minimum Value = 4 mA DC (From AI Module)" %
%   N24:2  AI_CURRENT_RANGE  "Analog Input Current Range Value = (AI_MAX - AI_MIN) For Use Elswhere" %
%   F26:133  FT03_25PCNT_VALUE  "FT-3 25% Range Value For HMI Display" %
%   F26:134  FT03_50PCNT_VALUE  "FT-3 50% Range Value For HMI Display" %
%   F26:135  FT03_75PCNT_VALUE  "FT-3 75% Range Value For HMI Display" %
%   F27:23  FT03_PID_FP  "FT-3 Flow Transmitter No-3 PID Statement Real Value" %
%   N24:22  PID_RANGE  "PID Statement Range Value = (PID_MAX - PID_MIN) For Use Elswhere" %
%   N24:20  PID_MIN  "PID Statement Minimum Value" %
%   N11:213  FT03_PID_MIN  "FT-3 Flow Transmitter No-3 PID Statement Minimum Input Value" %
%   N11:223  FT03_PID_MAX  "FT-3 Flow Transmitter No-3 PID Statement Maximum Input Value" %
%   N24:21  PID_MAX  "PID Statement Maximum Value" %
%   N11:203  FT03_PID_IN  "FT-3 Flow Transmitter No-3 PID Statement Input Value" %

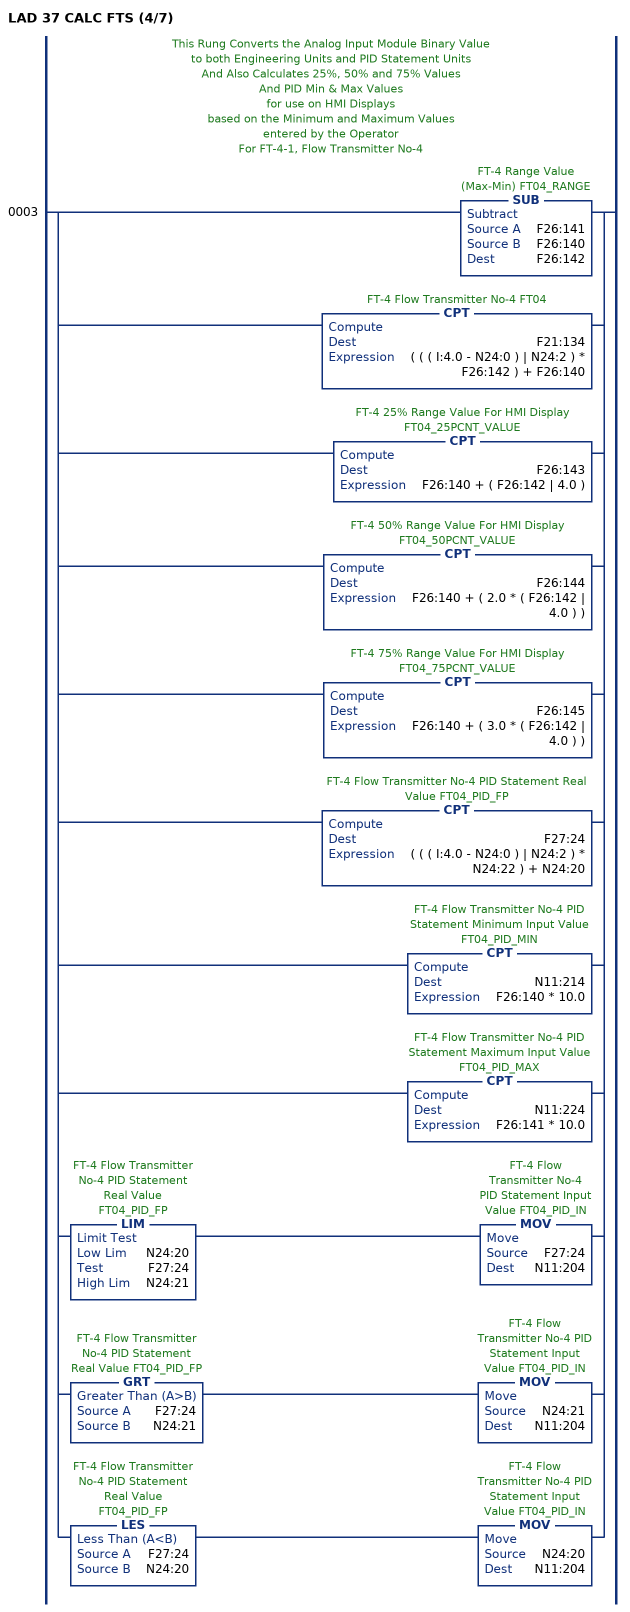
% Rung: 3 %
% This Rung Converts the Analog Input Module Binary Value
% to both Engineering Units and PID Statement Units
% And Also Calculates 25%, 50% and 75% Values
% And PID Min & Max Values
% for use on HMI Displays
% based on the Minimum and Maximum Values
% entered by the Operator
%    For FT-4-1, Flow Transmitter No-4 %
SOR BST SUB F26:141 F26:140 F26:142 NXB CPT F21:134 " ( ( ( I:4.0 - N24:0 ) | N24:2 ) * F26:142 ) + F26:140 " NXB CPT F26:143 " F26:140 + ( F26:142 | 4.0 ) " NXB CPT F26:144 " F26:140 + ( 2.0 * ( F26:142 | 4.0 ) ) " NXB CPT F26:145 " F26:140 + ( 3.0 * ( F26:142 | 4.0 ) ) " NXB CPT F27:24 " ( ( ( I:4.0 - N24:0 ) | N24:2 ) * N24:22 ) + N24:20 " NXB CPT N11:214 " F26:140 * 10.0 " NXB CPT N11:224 " F26:141 * 10.0 " NXB LIM N24:20 F27:24 N24:21 MOV F27:24 N11:204 NXB GRT F27:24 N24:21 MOV N24:21 N11:204 NXB LES F27:24 N24:20 MOV N24:20 N11:204 BND EOR
%   F26:141  FT04_MAX  "FT-4 Maximum Value" %
%   F26:140  FT04_MIN  "FT-4 Minimum Value" %
%   F26:142  FT04_RANGE  "FT-4 Range Value (Max-Min)" %
%   F21:134  FT04  "FT-4 Flow Transmitter No-4" %
%   I:4.0  FT04_BIN  "FT-4 Portable Mass Flowmeter Flow Signal No-4" %
%   N24:0  AI_CURRENT_MIN  "Analog Input Minimum Value = 4 mA DC (From AI Module)" %
%   N24:2  AI_CURRENT_RANGE  "Analog Input Current Range Value = (AI_MAX - AI_MIN) For Use Elswhere" %
%   F26:143  FT04_25PCNT_VALUE  "FT-4 25% Range Value For HMI Display" %
%   F26:144  FT04_50PCNT_VALUE  "FT-4 50% Range Value For HMI Display" %
%   F26:145  FT04_75PCNT_VALUE  "FT-4 75% Range Value For HMI Display" %
%   F27:24  FT04_PID_FP  "FT-4 Flow Transmitter No-4 PID Statement Real Value" %
%   N24:22  PID_RANGE  "PID Statement Range Value = (PID_MAX - PID_MIN) For Use Elswhere" %
%   N24:20  PID_MIN  "PID Statement Minimum Value" %
%   N11:214  FT04_PID_MIN  "FT-4 Flow Transmitter No-4 PID Statement Minimum Input Value" %
%   N11:224  FT04_PID_MAX  "FT-4 Flow Transmitter No-4 PID Statement Maximum Input Value" %
%   N24:21  PID_MAX  "PID Statement Maximum Value" %
%   N11:204  FT04_PID_IN  "FT-4 Flow Transmitter No-4 PID Statement Input Value" %

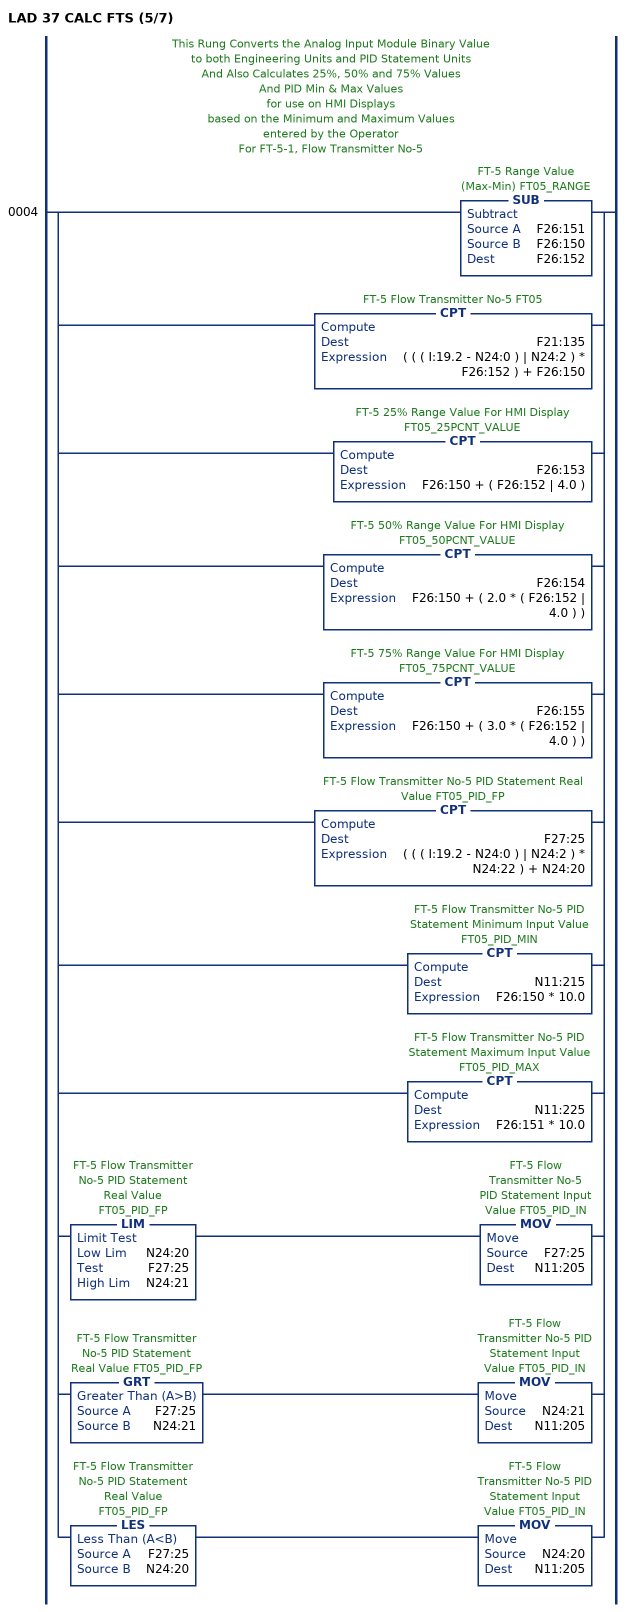
% Rung: 4 %
% This Rung Converts the Analog Input Module Binary Value
% to both Engineering Units and PID Statement Units
% And Also Calculates 25%, 50% and 75% Values
% And PID Min & Max Values
% for use on HMI Displays
% based on the Minimum and Maximum Values
% entered by the Operator
%    For FT-5-1, Flow Transmitter No-5 %
SOR BST SUB F26:151 F26:150 F26:152 NXB CPT F21:135 " ( ( ( I:19.2 - N24:0 ) | N24:2 ) * F26:152 ) + F26:150 " NXB CPT F26:153 " F26:150 + ( F26:152 | 4.0 ) " NXB CPT F26:154 " F26:150 + ( 2.0 * ( F26:152 | 4.0 ) ) " NXB CPT F26:155 " F26:150 + ( 3.0 * ( F26:152 | 4.0 ) ) " NXB CPT F27:25 " ( ( ( I:19.2 - N24:0 ) | N24:2 ) * N24:22 ) + N24:20 " NXB CPT N11:215 " F26:150 * 10.0 " NXB CPT N11:225 " F26:151 * 10.0 " NXB LIM N24:20 F27:25 N24:21 MOV F27:25 N11:205 NXB GRT F27:25 N24:21 MOV N24:21 N11:205 NXB LES F27:25 N24:20 MOV N24:20 N11:205 BND EOR
%   F26:151  FT05_MAX  "FT-5 Maximum Value" %
%   F26:150  FT05_MIN  "FT-5 Minimum Value" %
%   F26:152  FT05_RANGE  "FT-5 Range Value (Max-Min)" %
%   F21:135  FT05  "FT-5 Flow Transmitter No-5" %
%   I:19.2  FT05_BIN  "FT-5 Portable Mass Flowmeter Flow Signal No-5" %
%   N24:0  AI_CURRENT_MIN  "Analog Input Minimum Value = 4 mA DC (From AI Module)" %
%   N24:2  AI_CURRENT_RANGE  "Analog Input Current Range Value = (AI_MAX - AI_MIN) For Use Elswhere" %
%   F26:153  FT05_25PCNT_VALUE  "FT-5 25% Range Value For HMI Display" %
%   F26:154  FT05_50PCNT_VALUE  "FT-5 50% Range Value For HMI Display" %
%   F26:155  FT05_75PCNT_VALUE  "FT-5 75% Range Value For HMI Display" %
%   F27:25  FT05_PID_FP  "FT-5 Flow Transmitter No-5 PID Statement Real Value" %
%   N24:22  PID_RANGE  "PID Statement Range Value = (PID_MAX - PID_MIN) For Use Elswhere" %
%   N24:20  PID_MIN  "PID Statement Minimum Value" %
%   N11:215  FT05_PID_MIN  "FT-5 Flow Transmitter No-5 PID Statement Minimum Input Value" %
%   N11:225  FT05_PID_MAX  "FT-5 Flow Transmitter No-5 PID Statement Maximum Input Value" %
%   N24:21  PID_MAX  "PID Statement Maximum Value" %
%   N11:205  FT05_PID_IN  "FT-5 Flow Transmitter No-5 PID Statement Input Value" %

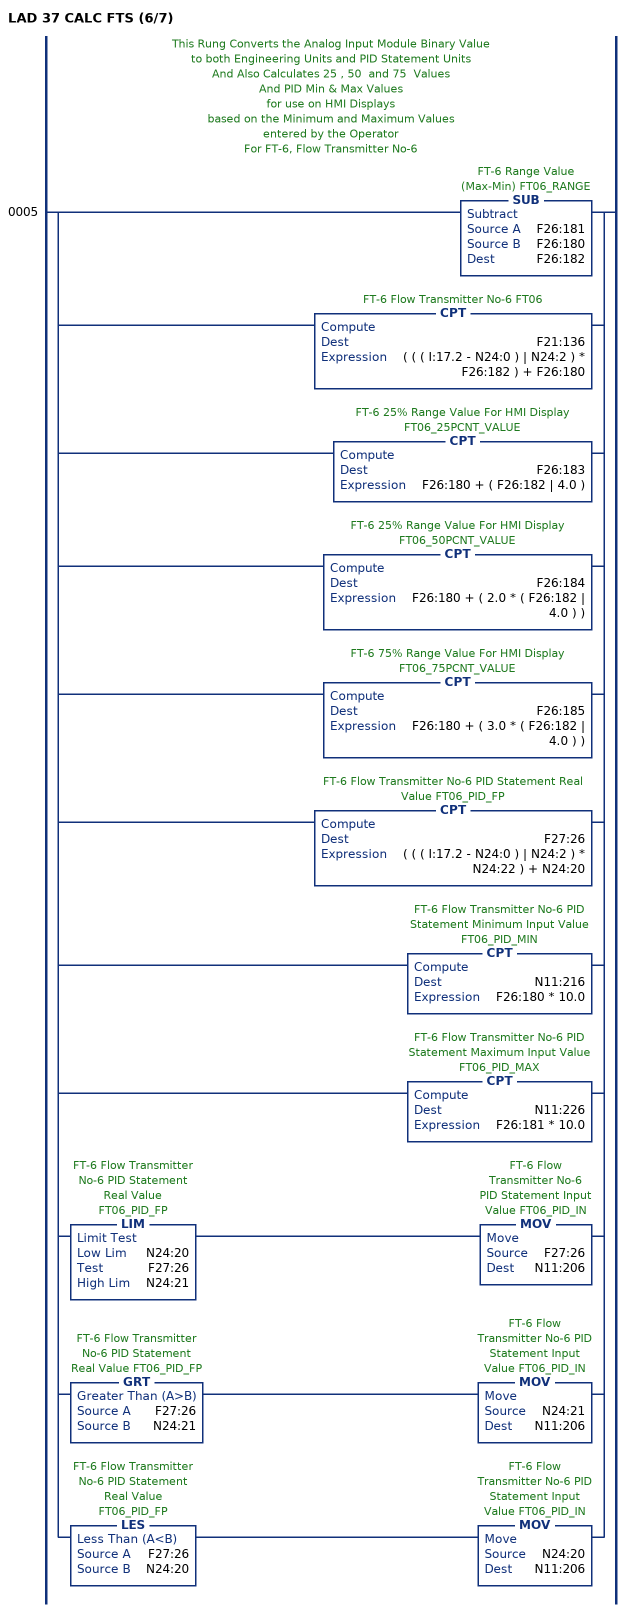
% Rung: 5 %
% This Rung Converts the Analog Input Module Binary Value
% to both Engineering Units and PID Statement Units
% And Also Calculates 25 , 50  and 75  Values
% And PID Min & Max Values
% for use on HMI Displays
% based on the Minimum and Maximum Values
% entered by the Operator
%    For FT-6, Flow Transmitter No-6 %
SOR BST SUB F26:181 F26:180 F26:182 NXB CPT F21:136 " ( ( ( I:17.2 - N24:0 ) | N24:2 ) * F26:182 ) + F26:180 " NXB CPT F26:183 " F26:180 + ( F26:182 | 4.0 ) " NXB CPT F26:184 " F26:180 + ( 2.0 * ( F26:182 | 4.0 ) ) " NXB CPT F26:185 " F26:180 + ( 3.0 * ( F26:182 | 4.0 ) ) " NXB CPT F27:26 " ( ( ( I:17.2 - N24:0 ) | N24:2 ) * N24:22 ) + N24:20 " NXB CPT N11:216 " F26:180 * 10.0 " NXB CPT N11:226 " F26:181 * 10.0 " NXB LIM N24:20 F27:26 N24:21 MOV F27:26 N11:206 NXB GRT F27:26 N24:21 MOV N24:21 N11:206 NXB LES F27:26 N24:20 MOV N24:20 N11:206 BND EOR
%   F26:181  FT06_MAX  "FT-6 Maximum Value" %
%   F26:180  FT06_MIN  "FT-6 Minimum Value" %
%   F26:182  FT06_RANGE  "FT-6 Range Value (Max-Min)" %
%   F21:136  FT06  "FT-6 Flow Transmitter No-6" %
%   I:17.2  FT06_BIN  "FT-6 Feed Flow Binary Input From Transmitter 1 Analog Input Module" %
%   N24:0  AI_CURRENT_MIN  "Analog Input Minimum Value = 4 mA DC (From AI Module)" %
%   N24:2  AI_CURRENT_RANGE  "Analog Input Current Range Value = (AI_MAX - AI_MIN) For Use Elswhere" %
%   F26:183  FT06_25PCNT_VALUE  "FT-6 25% Range Value For HMI Display" %
%   F26:184  FT06_50PCNT_VALUE  "FT-6 25% Range Value For HMI Display" %
%   F26:185  FT06_75PCNT_VALUE  "FT-6 75% Range Value For HMI Display" %
%   F27:26  FT06_PID_FP  "FT-6 Flow Transmitter No-6 PID Statement Real Value" %
%   N24:22  PID_RANGE  "PID Statement Range Value = (PID_MAX - PID_MIN) For Use Elswhere" %
%   N24:20  PID_MIN  "PID Statement Minimum Value" %
%   N11:216  FT06_PID_MIN  "FT-6 Flow Transmitter No-6 PID Statement Minimum Input Value" %
%   N11:226  FT06_PID_MAX  "FT-6 Flow Transmitter No-6 PID Statement Maximum Input Value" %
%   N24:21  PID_MAX  "PID Statement Maximum Value" %
%   N11:206  FT06_PID_IN  "FT-6 Flow Transmitter No-6 PID Statement Input Value" %

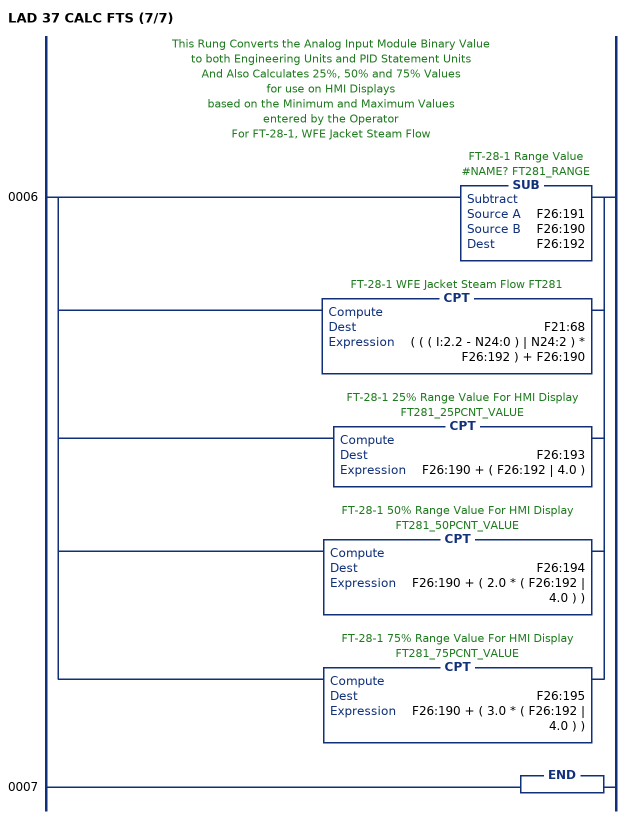
% Rung: 6 %
% This Rung Converts the Analog Input Module Binary Value
% to both Engineering Units and PID Statement Units
% And Also Calculates 25%, 50% and 75% Values
% for use on HMI Displays
% based on the Minimum and Maximum Values
% entered by the Operator
%    For FT-28-1, WFE Jacket Steam Flow %
SOR BST SUB F26:191 F26:190 F26:192 NXB CPT F21:68 " ( ( ( I:2.2 - N24:0 ) | N24:2 ) * F26:192 ) + F26:190 " NXB CPT F26:193 " F26:190 + ( F26:192 | 4.0 ) " NXB CPT F26:194 " F26:190 + ( 2.0 * ( F26:192 | 4.0 ) ) " NXB CPT F26:195 " F26:190 + ( 3.0 * ( F26:192 | 4.0 ) ) " BND EOR
%   F26:191  FT281_MAX  "FT-28-1 Maximum Value" %
%   F26:190  FT281_MIN  "FT-28-1 Minimum Value" %
%   F26:192  FT281_RANGE  "FT-28-1 Range Value #NAME?" %
%   F21:68  FT281  "FT-28-1 WFE Jacket Steam Flow" %
%   I:2.2  FT281_BIN  "FT-28-1 Steam Flow Binary Input From Transmitter Analog Input Module" %
%   N24:0  AI_CURRENT_MIN  "Analog Input Minimum Value = 4 mA DC (From AI Module)" %
%   N24:2  AI_CURRENT_RANGE  "Analog Input Current Range Value = (AI_MAX - AI_MIN) For Use Elswhere" %
%   F26:193  FT281_25PCNT_VALUE  "FT-28-1 25% Range Value For HMI Display" %
%   F26:194  FT281_50PCNT_VALUE  "FT-28-1 50% Range Value For HMI Display" %
%   F26:195  FT281_75PCNT_VALUE  "FT-28-1 75% Range Value For HMI Display" %
% Rung: 7 %
SOR END EOR

LADDER 38 "CALC FYS"    % Calculate Flow Rates based on Scale Change & Time %
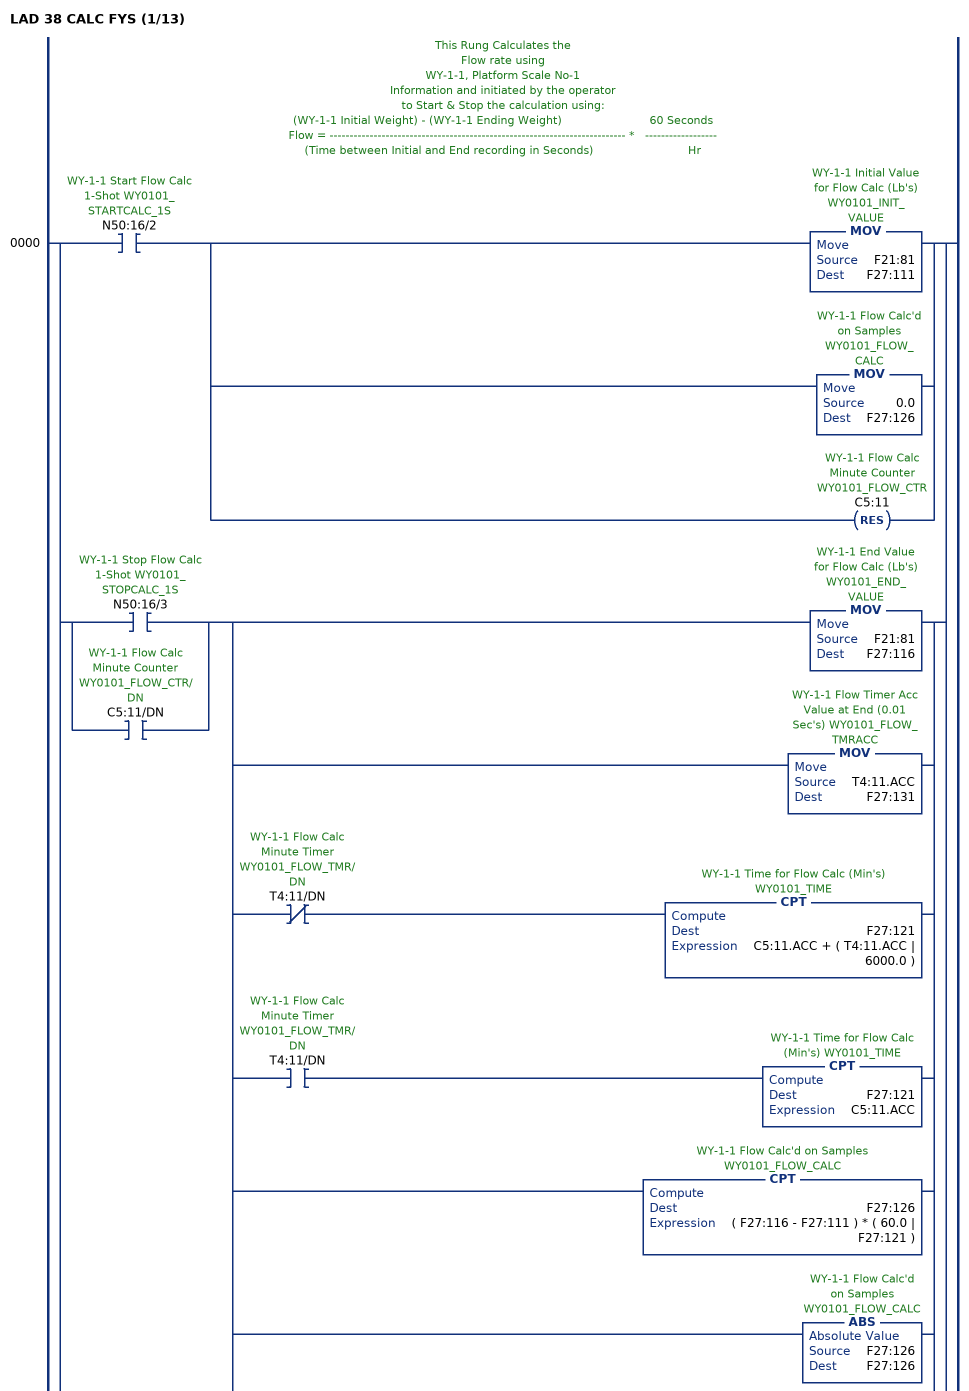
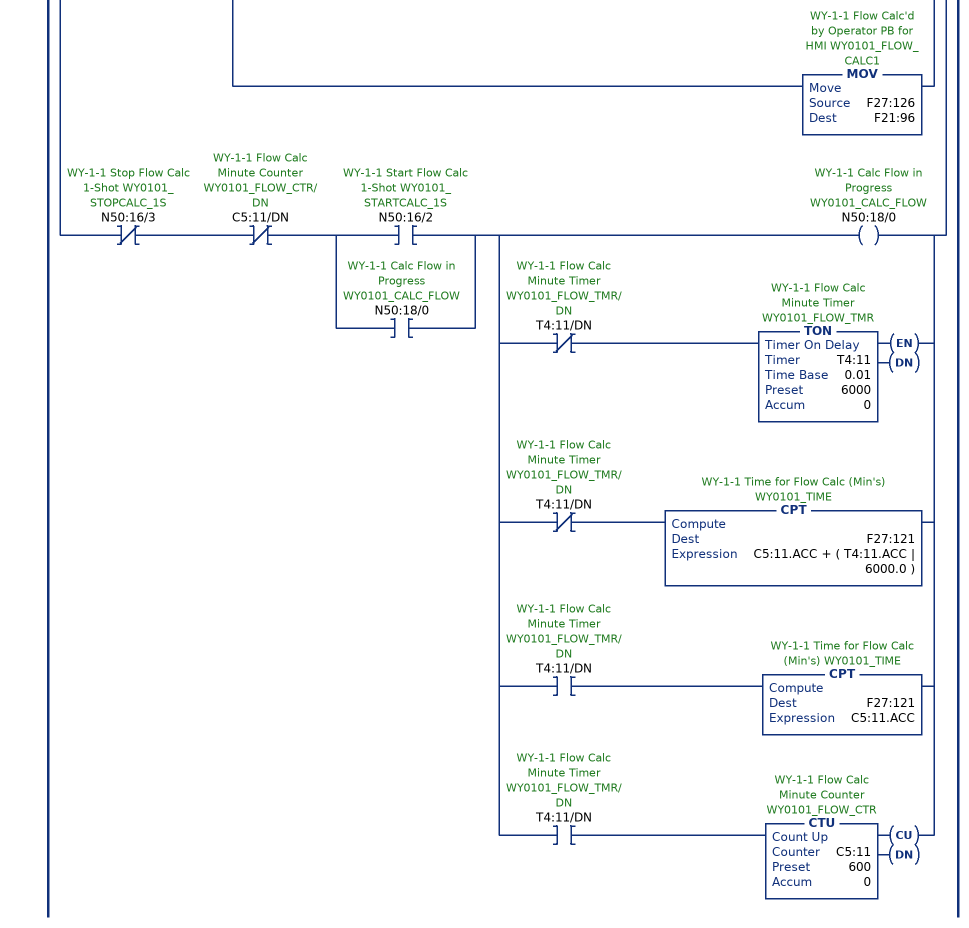
% Rung: 0 %
% This Rung Calculates the
% Flow rate using
% WY-1-1, Platform Scale No-1
% Information and initiated by the operator
% to Start & Stop the calculation using:
% 
%              (WY-1-1 Initial Weight) - (WY-1-1 Ending Weight)                         60 Seconds
% Flow = -------------------------------------------------------------------------- *   ------------------
%    (Time between Initial and End recording in Seconds)                           Hr %
SOR BST XIC N50:16/2 BST MOV F21:81 F27:111 NXB MOV 0.0 F27:126 NXB RES C5:11 BND NXB BST XIC N50:16/3 NXB XIC C5:11/DN BND BST MOV F21:81 F27:116 NXB MOV T4:11.ACC F27:131 NXB XIO T4:11/DN CPT F27:121 " C5:11.ACC + ( T4:11.ACC | 6000.0 ) " NXB XIC T4:11/DN CPT F27:121 "  C5:11.ACC " NXB CPT F27:126 " ( F27:116 - F27:111 ) * ( 60.0 | F27:121 ) " NXB ABS F27:126 F27:126 NXB MOV F27:126 F21:96 BND NXB XIO N50:16/3 XIO C5:11/DN BST XIC N50:16/2 NXB XIC N50:18/0 BND BST OTE N50:18/0 NXB XIO T4:11/DN TON T4:11 0.01 6000 0 NXB XIO T4:11/DN CPT F27:121 " C5:11.ACC + ( T4:11.ACC | 6000.0 ) " NXB XIC T4:11/DN CPT F27:121 "  C5:11.ACC " NXB XIC T4:11/DN CTU C5:11 600 0 BND BND EOR
%   N50:16/2  WY0101_STARTCALC_1S  "WY-1-1 Start Flow Calc 1-Shot" %
%   F21:81  WY0101  "WY-1-1 Platform Scale No-1 Weight" %
%   F27:111  WY0101_INIT_VALUE  "WY-1-1 Initial Value for Flow Calc (Lb's)" %
%   F27:126  WY0101_FLOW_CALC  "WY-1-1 Flow Calc'd on Samples" %
%   C5:11  WY0101_FLOW_CTR  "WY-1-1 Flow Calc Minute Counter" %
%   N50:16/3  WY0101_STOPCALC_1S  "WY-1-1 Stop Flow Calc 1-Shot" %
%   F27:116  WY0101_END_VALUE  "WY-1-1 End Value for Flow Calc (Lb's)" %
%   T4:11  WY0101_FLOW_TMR  "WY-1-1 Flow Calc Minute Timer" %
%   F27:131  WY0101_FLOW_TMRACC  "WY-1-1 Flow Timer Acc Value at End (0.01 Sec's)" %
%   F27:121  WY0101_TIME  "WY-1-1 Time for Flow Calc (Min's)" %
%   F21:96  WY0101_FLOW_CALC1  "WY-1-1 Flow Calc'd by Operator PB for HMI" %
%   N50:18/0  WY0101_CALC_FLOW  "WY-1-1 Calc Flow in Progress" %

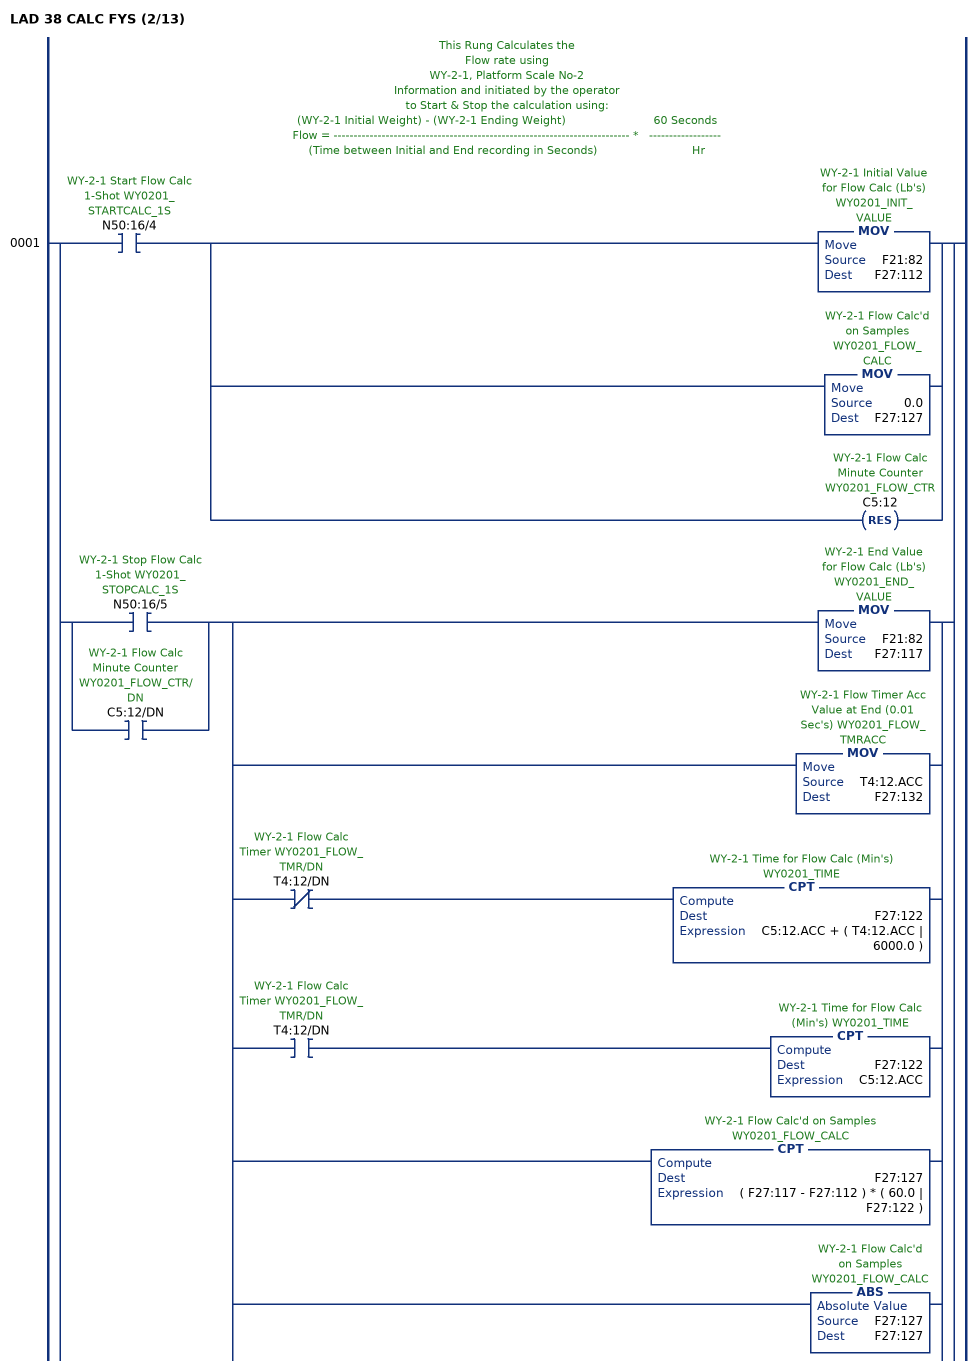

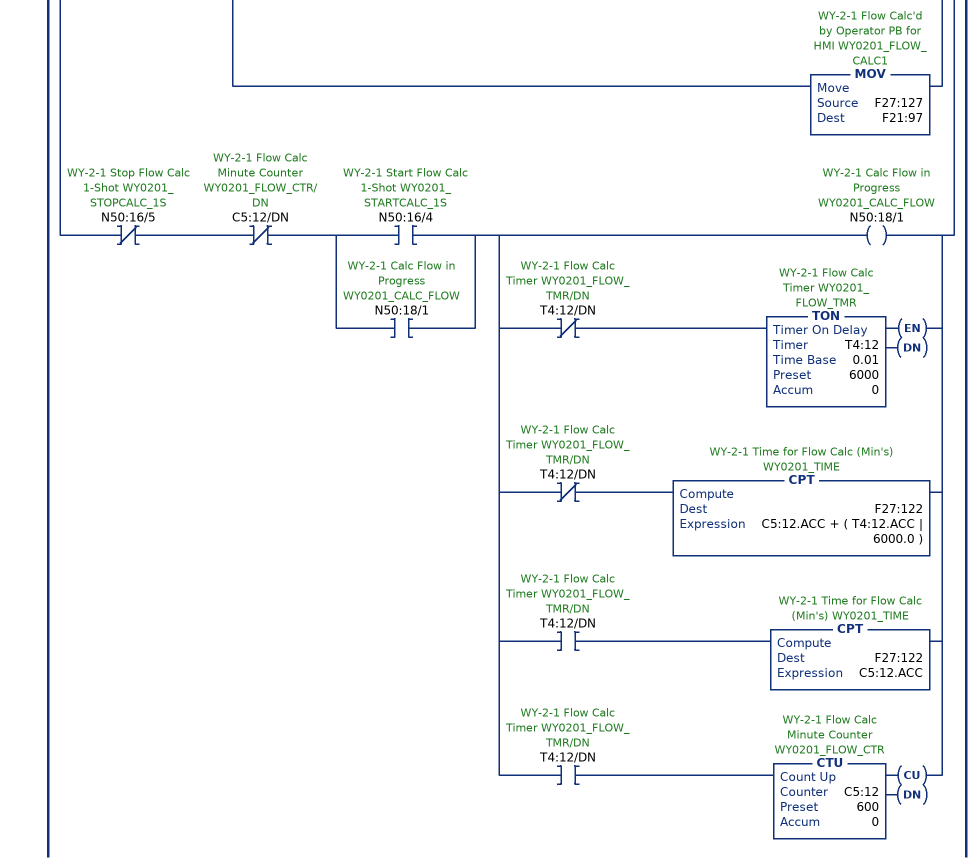
% Rung: 1 %
% This Rung Calculates the
% Flow rate using
% WY-2-1, Platform Scale No-2
% Information and initiated by the operator
% to Start & Stop the calculation using:
% 
%              (WY-2-1 Initial Weight) - (WY-2-1 Ending Weight)                         60 Seconds
% Flow = -------------------------------------------------------------------------- *   ------------------
%    (Time between Initial and End recording in Seconds)                           Hr %
SOR BST XIC N50:16/4 BST MOV F21:82 F27:112 NXB MOV 0.0 F27:127 NXB RES C5:12 BND NXB BST XIC N50:16/5 NXB XIC C5:12/DN BND BST MOV F21:82 F27:117 NXB MOV T4:12.ACC F27:132 NXB XIO T4:12/DN CPT F27:122 " C5:12.ACC + ( T4:12.ACC | 6000.0 ) " NXB XIC T4:12/DN CPT F27:122 "  C5:12.ACC " NXB CPT F27:127 " ( F27:117 - F27:112 ) * ( 60.0 | F27:122 ) " NXB ABS F27:127 F27:127 NXB MOV F27:127 F21:97 BND NXB XIO N50:16/5 XIO C5:12/DN BST XIC N50:16/4 NXB XIC N50:18/1 BND BST OTE N50:18/1 NXB XIO T4:12/DN TON T4:12 0.01 6000 0 NXB XIO T4:12/DN CPT F27:122 " C5:12.ACC + ( T4:12.ACC | 6000.0 ) " NXB XIC T4:12/DN CPT F27:122 "  C5:12.ACC " NXB XIC T4:12/DN CTU C5:12 600 0 BND BND EOR
%   N50:16/4  WY0201_STARTCALC_1S  "WY-2-1 Start Flow Calc 1-Shot" %
%   F21:82  WY0201  "WY-2-1 Platform Scale No-2 Weight" %
%   F27:112  WY0201_INIT_VALUE  "WY-2-1 Initial Value for Flow Calc (Lb's)" %
%   F27:127  WY0201_FLOW_CALC  "WY-2-1 Flow Calc'd on Samples" %
%   C5:12  WY0201_FLOW_CTR  "WY-2-1 Flow Calc Minute Counter" %
%   N50:16/5  WY0201_STOPCALC_1S  "WY-2-1 Stop Flow Calc 1-Shot" %
%   F27:117  WY0201_END_VALUE  "WY-2-1 End Value for Flow Calc (Lb's)" %
%   T4:12  WY0201_FLOW_TMR  "WY-2-1 Flow Calc Timer" %
%   F27:132  WY0201_FLOW_TMRACC  "WY-2-1 Flow Timer Acc Value at End (0.01 Sec's)" %
%   F27:122  WY0201_TIME  "WY-2-1 Time for Flow Calc (Min's)" %
%   F21:97  WY0201_FLOW_CALC1  "WY-2-1 Flow Calc'd by Operator PB for HMI" %
%   N50:18/1  WY0201_CALC_FLOW  "WY-2-1 Calc Flow in Progress" %

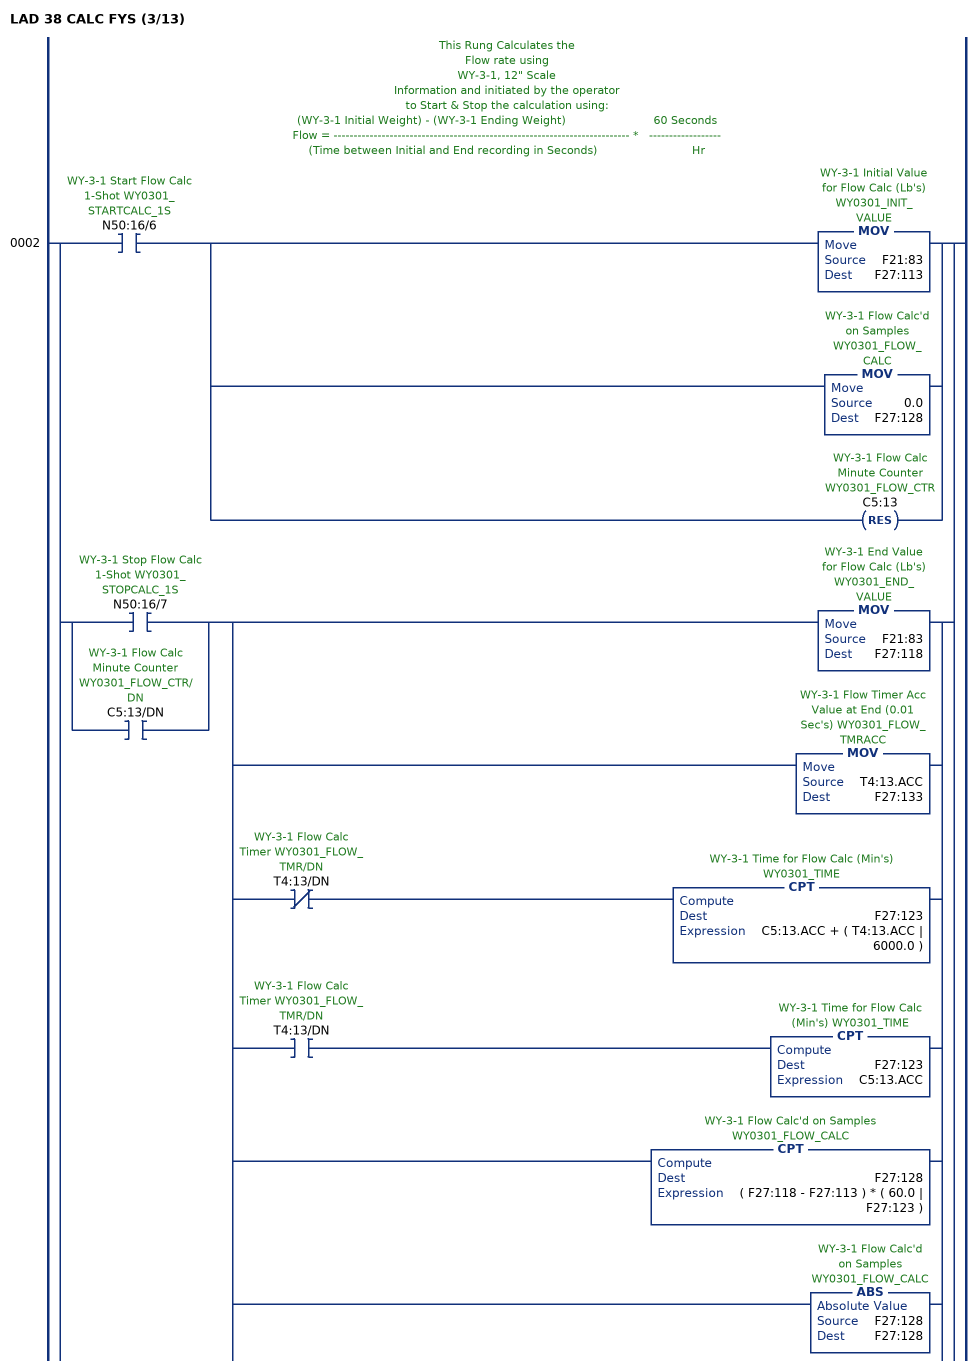

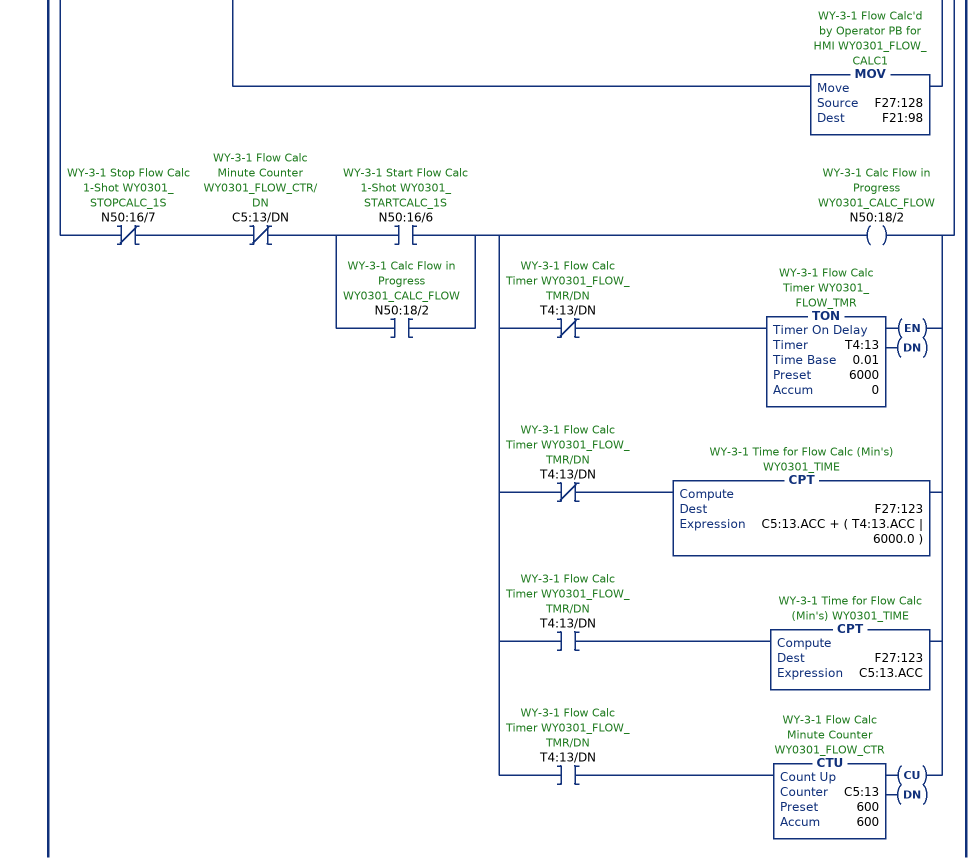
% Rung: 2 %
% This Rung Calculates the
% Flow rate using
% WY-3-1, 12" Scale
% Information and initiated by the operator
% to Start & Stop the calculation using:
% 
%              (WY-3-1 Initial Weight) - (WY-3-1 Ending Weight)                         60 Seconds
% Flow = -------------------------------------------------------------------------- *   ------------------
%    (Time between Initial and End recording in Seconds)                           Hr %
SOR BST XIC N50:16/6 BST MOV F21:83 F27:113 NXB MOV 0.0 F27:128 NXB RES C5:13 BND NXB BST XIC N50:16/7 NXB XIC C5:13/DN BND BST MOV F21:83 F27:118 NXB MOV T4:13.ACC F27:133 NXB XIO T4:13/DN CPT F27:123 " C5:13.ACC + ( T4:13.ACC | 6000.0 ) " NXB XIC T4:13/DN CPT F27:123 "  C5:13.ACC " NXB CPT F27:128 " ( F27:118 - F27:113 ) * ( 60.0 | F27:123 ) " NXB ABS F27:128 F27:128 NXB MOV F27:128 F21:98 BND NXB XIO N50:16/7 XIO C5:13/DN BST XIC N50:16/6 NXB XIC N50:18/2 BND BST OTE N50:18/2 NXB XIO T4:13/DN TON T4:13 0.01 6000 0 NXB XIO T4:13/DN CPT F27:123 " C5:13.ACC + ( T4:13.ACC | 6000.0 ) " NXB XIC T4:13/DN CPT F27:123 "  C5:13.ACC " NXB XIC T4:13/DN CTU C5:13 600 600 BND BND EOR
%   N50:16/6  WY0301_STARTCALC_1S  "WY-3-1 Start Flow Calc 1-Shot" %
%   F21:83  WY0301  "WY-3-1 Platform Scale No-3 Weight 12" x 12" Scale" %
%   F27:113  WY0301_INIT_VALUE  "WY-3-1 Initial Value for Flow Calc (Lb's)" %
%   F27:128  WY0301_FLOW_CALC  "WY-3-1 Flow Calc'd on Samples" %
%   C5:13  WY0301_FLOW_CTR  "WY-3-1 Flow Calc Minute Counter" %
%   N50:16/7  WY0301_STOPCALC_1S  "WY-3-1 Stop Flow Calc 1-Shot" %
%   F27:118  WY0301_END_VALUE  "WY-3-1 End Value for Flow Calc (Lb's)" %
%   T4:13  WY0301_FLOW_TMR  "WY-3-1 Flow Calc Timer" %
%   F27:133  WY0301_FLOW_TMRACC  "WY-3-1 Flow Timer Acc Value at End (0.01 Sec's)" %
%   F27:123  WY0301_TIME  "WY-3-1 Time for Flow Calc (Min's)" %
%   F21:98  WY0301_FLOW_CALC1  "WY-3-1 Flow Calc'd by Operator PB for HMI" %
%   N50:18/2  WY0301_CALC_FLOW  "WY-3-1 Calc Flow in Progress" %

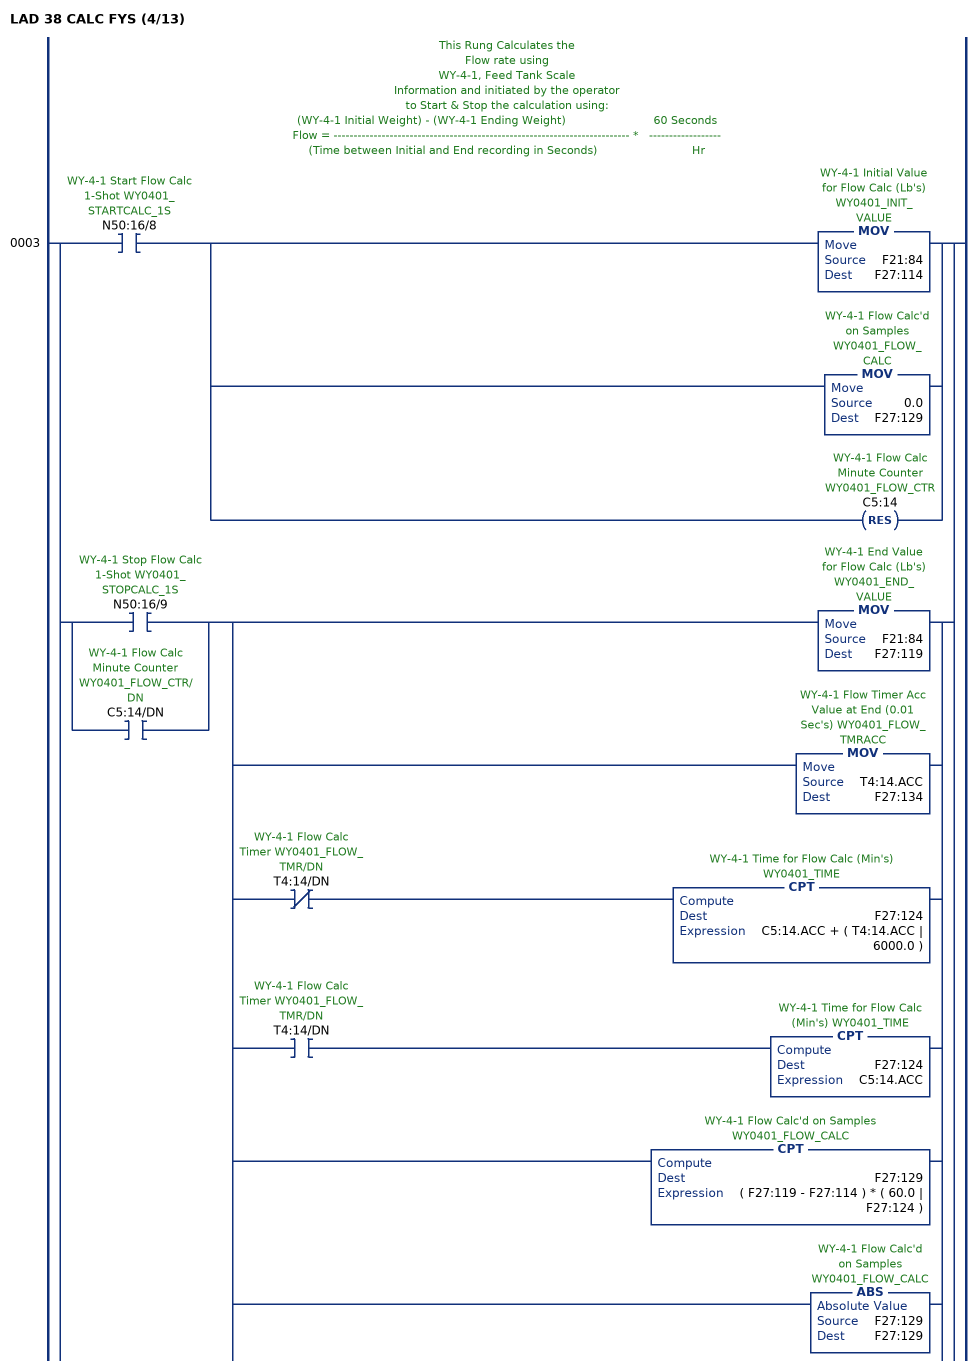

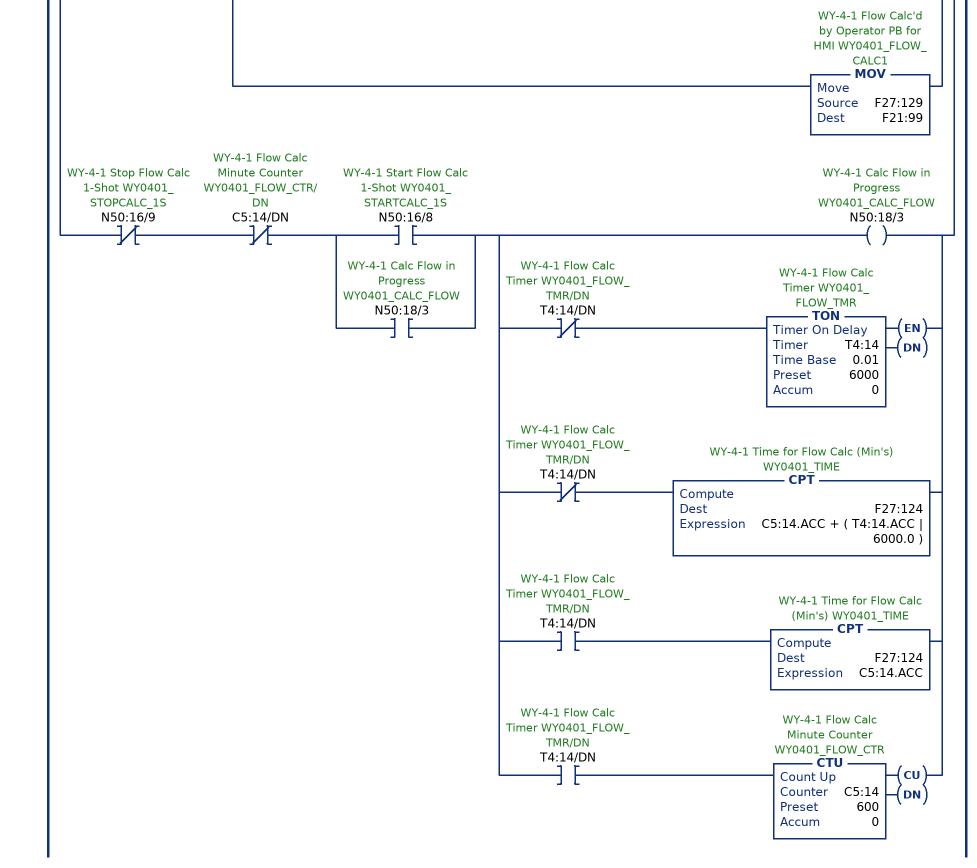
% Rung: 3 %
% This Rung Calculates the
% Flow rate using
% WY-4-1, Feed Tank Scale
% Information and initiated by the operator
% to Start & Stop the calculation using:
% 
%              (WY-4-1 Initial Weight) - (WY-4-1 Ending Weight)                         60 Seconds
% Flow = -------------------------------------------------------------------------- *   ------------------
%    (Time between Initial and End recording in Seconds)                           Hr %
SOR BST XIC N50:16/8 BST MOV F21:84 F27:114 NXB MOV 0.0 F27:129 NXB RES C5:14 BND NXB BST XIC N50:16/9 NXB XIC C5:14/DN BND BST MOV F21:84 F27:119 NXB MOV T4:14.ACC F27:134 NXB XIO T4:14/DN CPT F27:124 " C5:14.ACC + ( T4:14.ACC | 6000.0 ) " NXB XIC T4:14/DN CPT F27:124 "  C5:14.ACC " NXB CPT F27:129 " ( F27:119 - F27:114 ) * ( 60.0 | F27:124 ) " NXB ABS F27:129 F27:129 NXB MOV F27:129 F21:99 BND NXB XIO N50:16/9 XIO C5:14/DN BST XIC N50:16/8 NXB XIC N50:18/3 BND BST OTE N50:18/3 NXB XIO T4:14/DN TON T4:14 0.01 6000 0 NXB XIO T4:14/DN CPT F27:124 " C5:14.ACC + ( T4:14.ACC | 6000.0 ) " NXB XIC T4:14/DN CPT F27:124 "  C5:14.ACC " NXB XIC T4:14/DN CTU C5:14 600 0 BND BND EOR
%   N50:16/8  WY0401_STARTCALC_1S  "WY-4-1 Start Flow Calc 1-Shot" %
%   F21:84  WY0401  "WY-4-1 Feed Tank Weight" %
%   F27:114  WY0401_INIT_VALUE  "WY-4-1 Initial Value for Flow Calc (Lb's)" %
%   F27:129  WY0401_FLOW_CALC  "WY-4-1 Flow Calc'd on Samples" %
%   C5:14  WY0401_FLOW_CTR  "WY-4-1 Flow Calc Minute Counter" %
%   N50:16/9  WY0401_STOPCALC_1S  "WY-4-1 Stop Flow Calc 1-Shot" %
%   F27:119  WY0401_END_VALUE  "WY-4-1 End Value for Flow Calc (Lb's)" %
%   T4:14  WY0401_FLOW_TMR  "WY-4-1 Flow Calc Timer" %
%   F27:134  WY0401_FLOW_TMRACC  "WY-4-1 Flow Timer Acc Value at End (0.01 Sec's)" %
%   F27:124  WY0401_TIME  "WY-4-1 Time for Flow Calc (Min's)" %
%   F21:99  WY0401_FLOW_CALC1  "WY-4-1 Flow Calc'd by Operator PB for HMI" %
%   N50:18/3  WY0401_CALC_FLOW  "WY-4-1 Calc Flow in Progress" %

